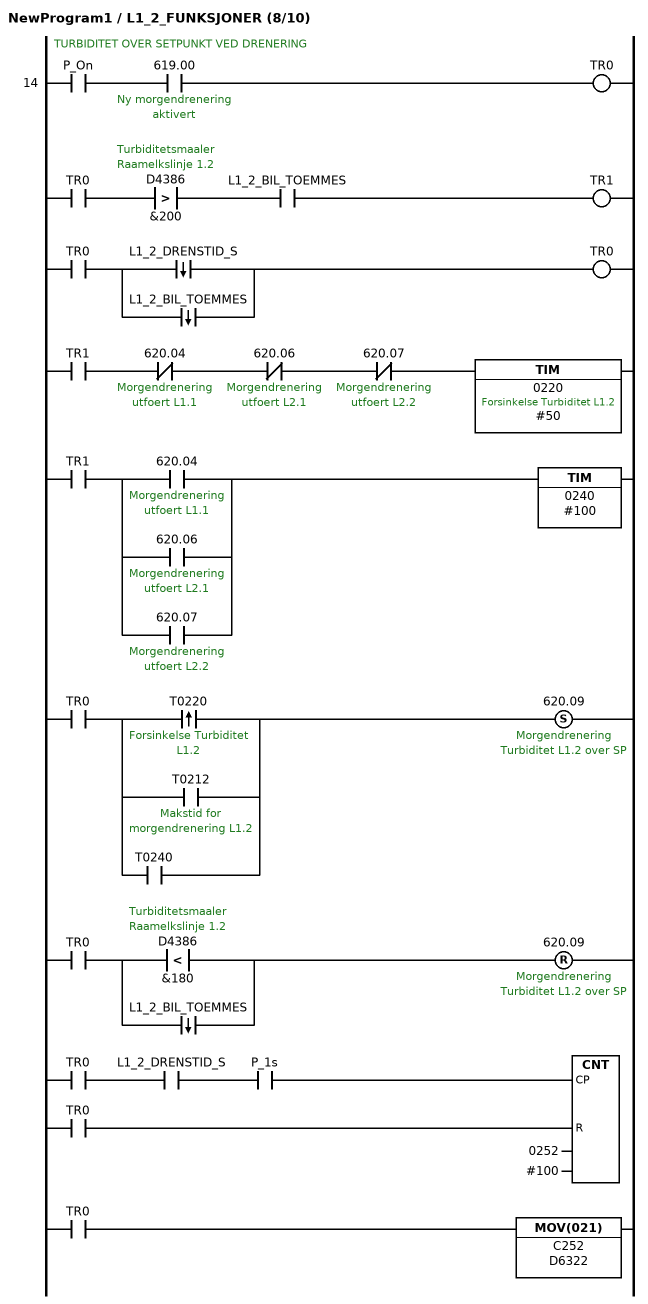
; [picture p792: NewProgram1 / L1_2_FUNKSJONER, rungs 14-14]
; rung 14: TURBIDITET OVER SETPUNKT VED DRENERING
LD P_On
AND 619.00  ; Ny morgendrenering aktivert
OUT TR0
AND>(320) D4386 &200  ; Turbiditetsmaaler Raamelkslinje 1.2
AND L1_2_BIL_TOEMMES
OUT TR1
ANDNOT 620.04  ; Morgendrenering utfoert L1.1
ANDNOT 620.06  ; Morgendrenering utfoert L2.1
ANDNOT 620.07  ; Morgendrenering utfoert L2.2
TIM 0220 #50  ; Forsinkelse Turbiditet L1.2
LD TR1
LD 620.04  ; Morgendrenering utfoert L1.1
OR 620.06  ; Morgendrenering utfoert L2.1
OR 620.07  ; Morgendrenering utfoert L2.2
ANDLD
TIM 0240 #100
LD TR0
@LD T0220  ; Forsinkelse Turbiditet L1.2
OR T0212  ; Makstid for morgendrenering L1.2
OR T0240
ANDLD
SET 620.09  ; Morgendrenering Turbiditet L1.2 over SP
LD TR0
LD<(310) D4386 &180  ; Turbiditetsmaaler Raamelkslinje 1.2
%OR L1_2_BIL_TOEMMES
ANDLD
RSET 620.09  ; Morgendrenering Turbiditet L1.2 over SP
LD TR0
AND L1_2_DRENSTID_S
AND P_1s
LD TR0
%LD L1_2_DRENSTID_S
%OR L1_2_BIL_TOEMMES
ANDLD
OUT TR0
CNT 0252 #100
LD TR0
MOV(021) C252 D6322

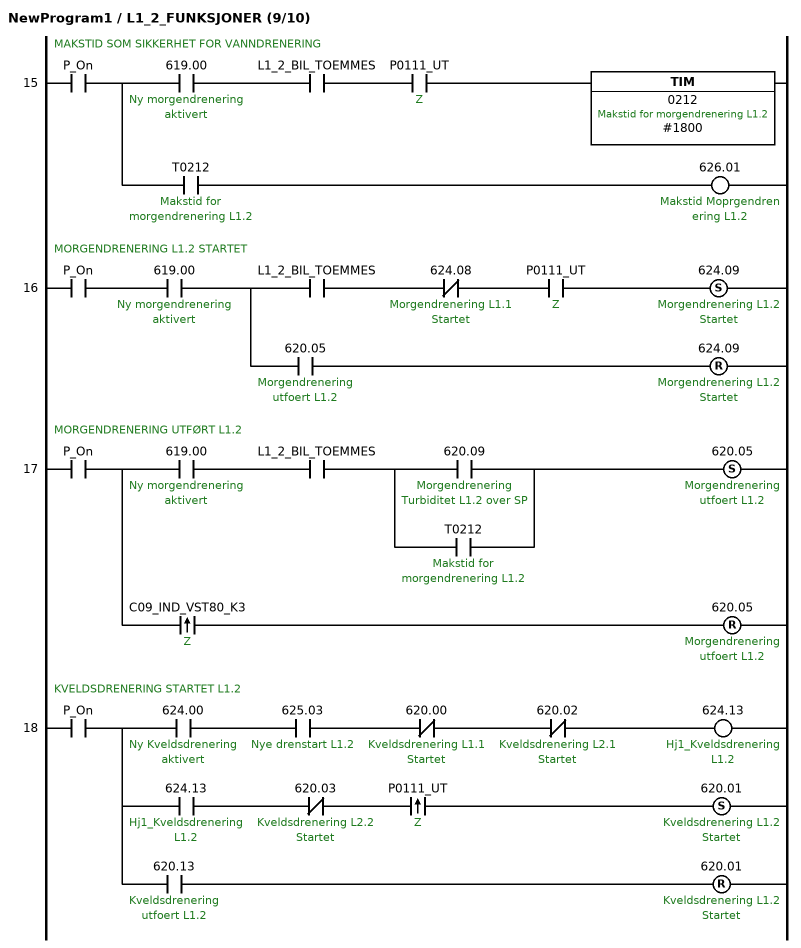
; rung 15: MAKSTID SOM SIKKERHET FOR VANNDRENERING
LD P_On
OUT TR0
AND 619.00  ; Ny morgendrenering aktivert
AND L1_2_BIL_TOEMMES
AND P0111_UT  ; Z
TIM 0212 #1800  ; Makstid for morgendrenering L1.2
LD TR0
AND T0212  ; Makstid for morgendrenering L1.2
OUT 626.01  ; Makstid Moprgendrenering L1.2
; rung 16: MORGENDRENERING L1.2 STARTET
LD P_On
AND 619.00  ; Ny morgendrenering aktivert
OUT TR0
AND L1_2_BIL_TOEMMES
ANDNOT 624.08  ; Morgendrenering L1.1 Startet
AND P0111_UT  ; Z
SET 624.09  ; Morgendrenering L1.2 Startet
LD TR0
AND 620.05  ; Morgendrenering utfoert L1.2
RSET 624.09  ; Morgendrenering L1.2 Startet
; rung 17: MORGENDRENERING UTFØRT L1.2
LD P_On
OUT TR0
AND 619.00  ; Ny morgendrenering aktivert
AND L1_2_BIL_TOEMMES
LD 620.09  ; Morgendrenering Turbiditet L1.2 over SP
OR T0212  ; Makstid for morgendrenering L1.2
ANDLD
SET 620.05  ; Morgendrenering utfoert L1.2
LD TR0
@AND C09_IND_VST80_K3  ; Z
RSET 620.05  ; Morgendrenering utfoert L1.2
; rung 18: KVELDSDRENERING STARTET L1.2
LD P_On
OUT TR0
AND 624.00  ; Ny Kveldsdrenering aktivert
AND 625.03  ; Nye drenstart L1.2
ANDNOT 620.00  ; Kveldsdrenering L1.1 Startet
ANDNOT 620.02  ; Kveldsdrenering L2.1 Startet
OUT 624.13  ; Hj1_Kveldsdrenering L1.2
LD TR0
AND 624.13  ; Hj1_Kveldsdrenering L1.2
ANDNOT 620.03  ; Kveldsdrenering L2.2 Startet
@AND P0111_UT  ; Z
SET 620.01  ; Kveldsdrenering L1.2 Startet
LD TR0
AND 620.13  ; Kveldsdrenering utfoert L1.2
RSET 620.01  ; Kveldsdrenering L1.2 Startet

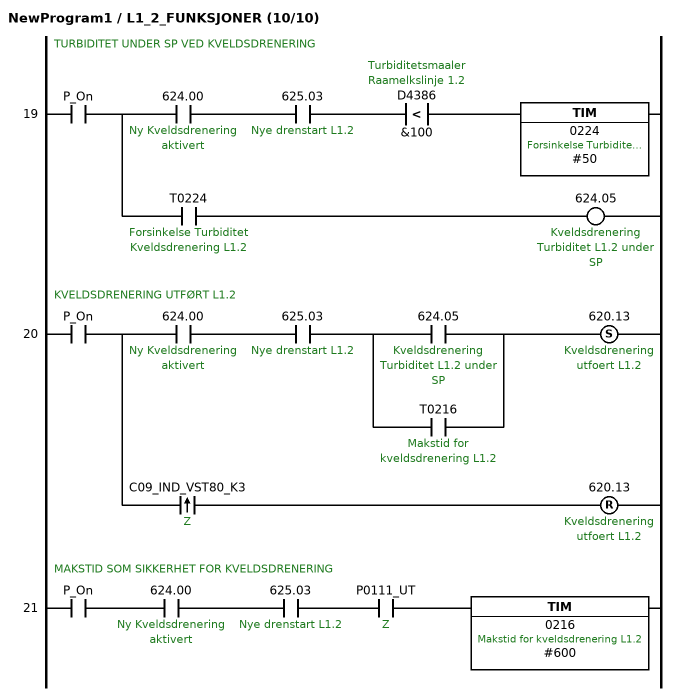
; rung 19: TURBIDITET UNDER SP VED KVELDSDRENERING
LD P_On
OUT TR0
AND 624.00  ; Ny Kveldsdrenering aktivert
AND 625.03  ; Nye drenstart L1.2
AND<(310) D4386 &100  ; Turbiditetsmaaler Raamelkslinje 1.2
TIM 0224 #50  ; Forsinkelse Turbiditet Kveldsdrenering L1.2
LD TR0
AND T0224  ; Forsinkelse Turbiditet Kveldsdrenering L1.2
OUT 624.05  ; Kveldsdrenering Turbiditet L1.2 under SP
; rung 20: KVELDSDRENERING UTFØRT L1.2
LD P_On
OUT TR0
AND 624.00  ; Ny Kveldsdrenering aktivert
AND 625.03  ; Nye drenstart L1.2
LD 624.05  ; Kveldsdrenering Turbiditet L1.2 under SP
OR T0216  ; Makstid for kveldsdrenering L1.2
ANDLD
SET 620.13  ; Kveldsdrenering utfoert L1.2
LD TR0
@AND C09_IND_VST80_K3  ; Z
RSET 620.13  ; Kveldsdrenering utfoert L1.2
; rung 21: MAKSTID SOM SIKKERHET FOR KVELDSDRENERING
LD P_On
AND 624.00  ; Ny Kveldsdrenering aktivert
AND 625.03  ; Nye drenstart L1.2
AND P0111_UT  ; Z
TIM 0216 #600  ; Makstid for kveldsdrenering L1.2
; rung 22: Ingen_kommentar_funnet

### Section L2_1_STATUS

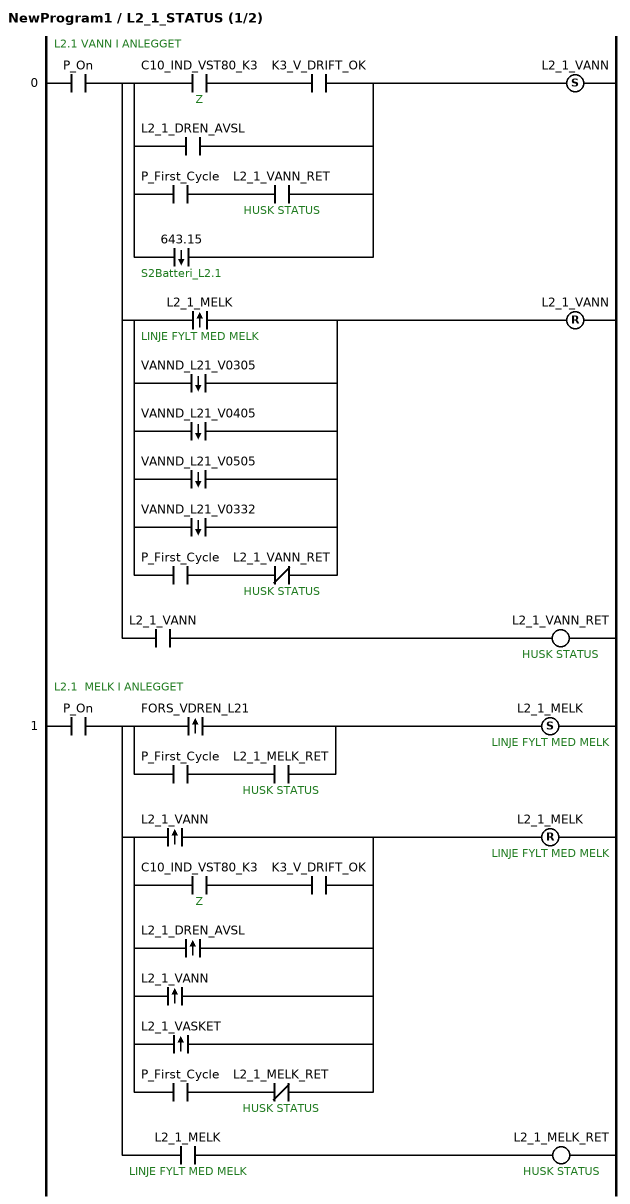
; rung 0: L2.1 VANN I ANLEGGET
LD P_On
OUT TR0
LD C10_IND_VST80_K3  ; Z
AND K3_V_DRIFT_OK
OR L2_1_DREN_AVSL
LD P_First_Cycle
AND L2_1_VANN_RET  ; HUSK STATUS
ORLD
%OR 643.15  ; S2Batteri_L2.1
ANDLD
SET L2_1_VANN
LD TR0
@LD L2_1_MELK  ; LINJE FYLT MED MELK
%OR VANND_L21_V0305
%OR VANND_L21_V0405
%OR VANND_L21_V0505
%OR VANND_L21_V0332
LD P_First_Cycle
ANDNOT L2_1_VANN_RET  ; HUSK STATUS
ORLD
ANDLD
RSET L2_1_VANN
LD TR0
AND L2_1_VANN
OUT L2_1_VANN_RET  ; HUSK STATUS
; rung 1: L2.1  MELK I ANLEGGET
LD P_On
OUT TR0
@LD FORS_VDREN_L21
LD P_First_Cycle
AND L2_1_MELK_RET  ; HUSK STATUS
ORLD
ANDLD
SET L2_1_MELK  ; LINJE FYLT MED MELK
LD TR0
@LD L2_1_VANN
LD C10_IND_VST80_K3  ; Z
AND K3_V_DRIFT_OK
ORLD
@OR L2_1_DREN_AVSL
@OR L2_1_VANN
@OR L2_1_VASKET
LD P_First_Cycle
ANDNOT L2_1_MELK_RET  ; HUSK STATUS
ORLD
ANDLD
RSET L2_1_MELK  ; LINJE FYLT MED MELK
LD TR0
AND L2_1_MELK  ; LINJE FYLT MED MELK
OUT L2_1_MELK_RET  ; HUSK STATUS

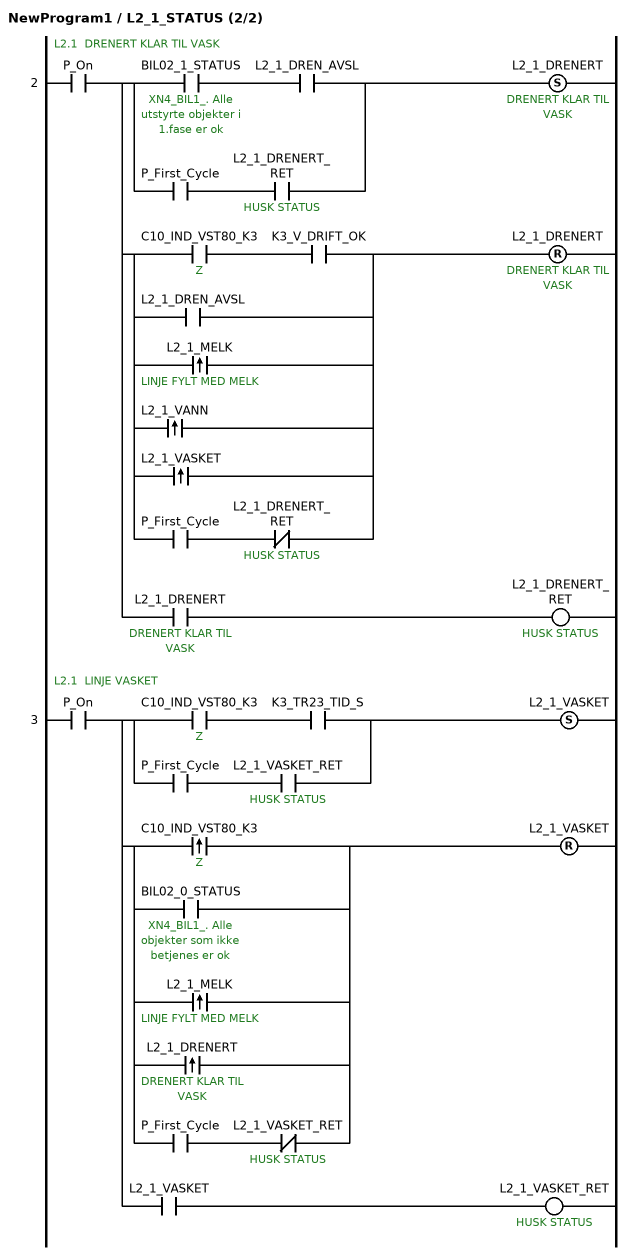
; rung 2: L2.1  DRENERT KLAR TIL VASK
LD P_On
OUT TR0
LD BIL02_1_STATUS  ; XN4_BIL1_. Alle utstyrte objekter i 1.fase er ok
AND L2_1_DREN_AVSL
LD P_First_Cycle
AND L2_1_DRENERT_RET  ; HUSK STATUS
ORLD
ANDLD
SET L2_1_DRENERT  ; DRENERT KLAR TIL VASK
LD TR0
LD C10_IND_VST80_K3  ; Z
AND K3_V_DRIFT_OK
OR L2_1_DREN_AVSL
@OR L2_1_MELK  ; LINJE FYLT MED MELK
@OR L2_1_VANN
@OR L2_1_VASKET
LD P_First_Cycle
ANDNOT L2_1_DRENERT_RET  ; HUSK STATUS
ORLD
ANDLD
RSET L2_1_DRENERT  ; DRENERT KLAR TIL VASK
LD TR0
AND L2_1_DRENERT  ; DRENERT KLAR TIL VASK
OUT L2_1_DRENERT_RET  ; HUSK STATUS
; rung 3: L2.1  LINJE VASKET
LD P_On
OUT TR0
LD C10_IND_VST80_K3  ; Z
AND K3_TR23_TID_S
LD P_First_Cycle
AND L2_1_VASKET_RET  ; HUSK STATUS
ORLD
ANDLD
SET L2_1_VASKET
LD TR0
@LD C10_IND_VST80_K3  ; Z
OR BIL02_0_STATUS  ; XN4_BIL1_. Alle objekter som ikke betjenes er ok
@OR L2_1_MELK  ; LINJE FYLT MED MELK
@OR L2_1_DRENERT  ; DRENERT KLAR TIL VASK
LD P_First_Cycle
ANDNOT L2_1_VASKET_RET  ; HUSK STATUS
ORLD
ANDLD
RSET L2_1_VASKET
LD TR0
AND L2_1_VASKET
OUT L2_1_VASKET_RET  ; HUSK STATUS
; rung 4: Ingen_kommentar_funnet

### Section L1_1_L1_2_FELLESFUNKSJONER

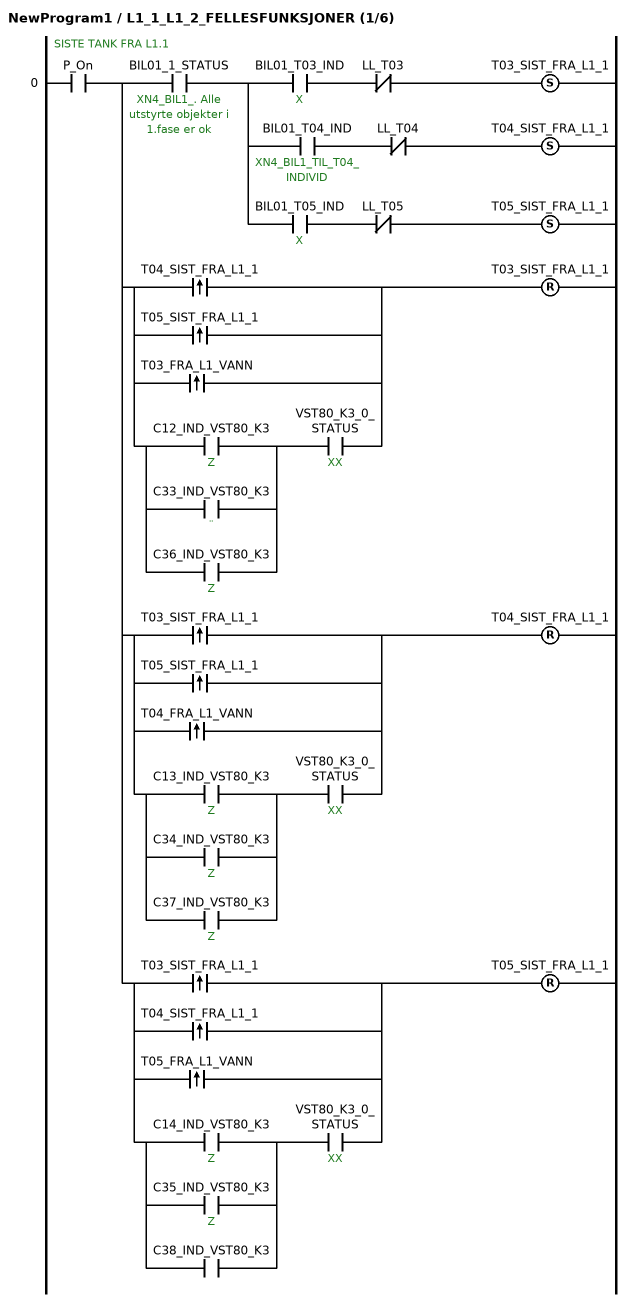
; rung 0: SISTE TANK FRA L1.1
LD P_On
OUT TR0
AND BIL01_1_STATUS  ; XN4_BIL1_. Alle utstyrte objekter i 1.fase er ok
OUT TR1
AND BIL01_T03_IND  ; X
ANDNOT LL_T03
SET T03_SIST_FRA_L1_1
LD TR1
AND BIL01_T04_IND  ; XN4_BIL1_TIL_T04_INDIVID
ANDNOT LL_T04
SET T04_SIST_FRA_L1_1
LD TR1
AND BIL01_T05_IND  ; X
ANDNOT LL_T05
SET T05_SIST_FRA_L1_1
LD TR0
@LD T04_SIST_FRA_L1_1
@OR T05_SIST_FRA_L1_1
@OR T03_FRA_L1_VANN
LD C12_IND_VST80_K3  ; Z
OR C33_IND_VST80_K3  ; ¨
OR C36_IND_VST80_K3  ; Z
AND VST80_K3_0_STATUS  ; XX
ORLD
ANDLD
RSET T03_SIST_FRA_L1_1
LD TR0
@LD T03_SIST_FRA_L1_1
@OR T05_SIST_FRA_L1_1
@OR T04_FRA_L1_VANN
LD C13_IND_VST80_K3  ; Z
OR C34_IND_VST80_K3  ; Z
OR C37_IND_VST80_K3  ; Z
AND VST80_K3_0_STATUS  ; XX
ORLD
ANDLD
RSET T04_SIST_FRA_L1_1
LD TR0
@LD T03_SIST_FRA_L1_1
@OR T04_SIST_FRA_L1_1
@OR T05_FRA_L1_VANN
LD C14_IND_VST80_K3  ; Z
OR C35_IND_VST80_K3  ; Z
OR C38_IND_VST80_K3
AND VST80_K3_0_STATUS  ; XX
ORLD
ANDLD
RSET T05_SIST_FRA_L1_1

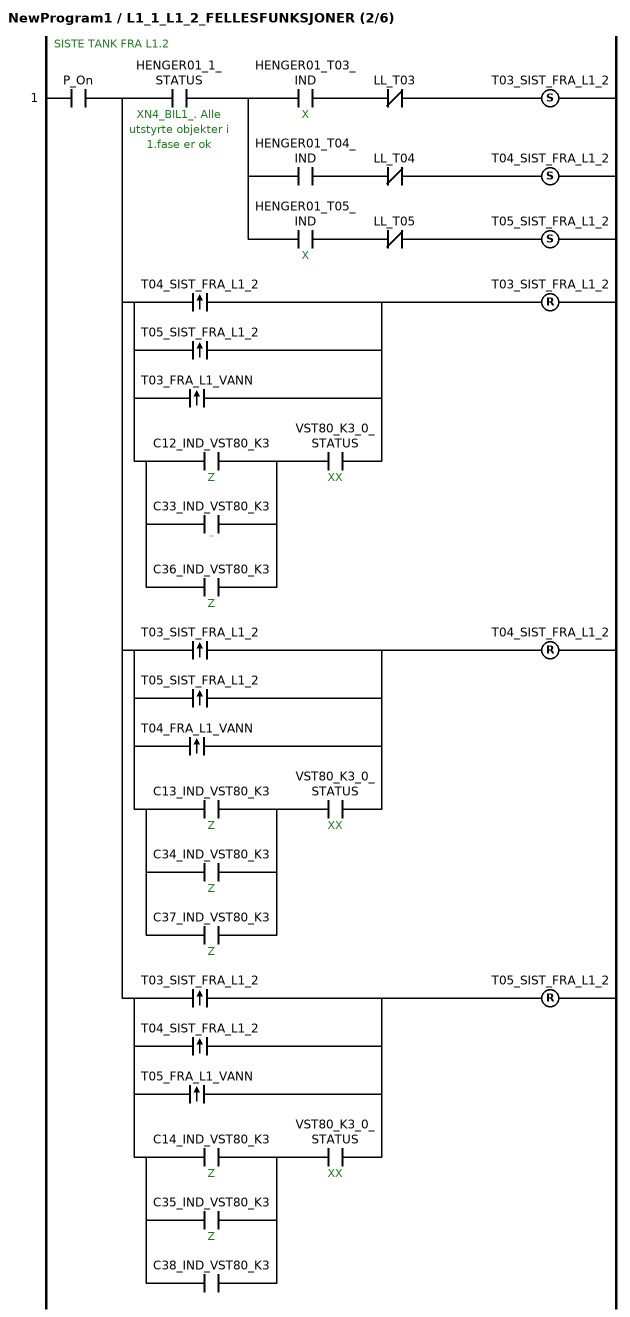
; rung 1: SISTE TANK FRA L1.2
LD P_On
OUT TR0
AND HENGER01_1_STATUS  ; XN4_BIL1_. Alle utstyrte objekter i 1.fase er ok
OUT TR1
AND HENGER01_T03_IND  ; X
ANDNOT LL_T03
SET T03_SIST_FRA_L1_2
LD TR1
AND HENGER01_T04_IND
ANDNOT LL_T04
SET T04_SIST_FRA_L1_2
LD TR1
AND HENGER01_T05_IND  ; X
ANDNOT LL_T05
SET T05_SIST_FRA_L1_2
LD TR0
@LD T04_SIST_FRA_L1_2
@OR T05_SIST_FRA_L1_2
@OR T03_FRA_L1_VANN
LD C12_IND_VST80_K3  ; Z
OR C33_IND_VST80_K3  ; ¨
OR C36_IND_VST80_K3  ; Z
AND VST80_K3_0_STATUS  ; XX
ORLD
ANDLD
RSET T03_SIST_FRA_L1_2
LD TR0
@LD T03_SIST_FRA_L1_2
@OR T05_SIST_FRA_L1_2
@OR T04_FRA_L1_VANN
LD C13_IND_VST80_K3  ; Z
OR C34_IND_VST80_K3  ; Z
OR C37_IND_VST80_K3  ; Z
AND VST80_K3_0_STATUS  ; XX
ORLD
ANDLD
RSET T04_SIST_FRA_L1_2
LD TR0
@LD T03_SIST_FRA_L1_2
@OR T04_SIST_FRA_L1_2
@OR T05_FRA_L1_VANN
LD C14_IND_VST80_K3  ; Z
OR C35_IND_VST80_K3  ; Z
OR C38_IND_VST80_K3
AND VST80_K3_0_STATUS  ; XX
ORLD
ANDLD
RSET T05_SIST_FRA_L1_2

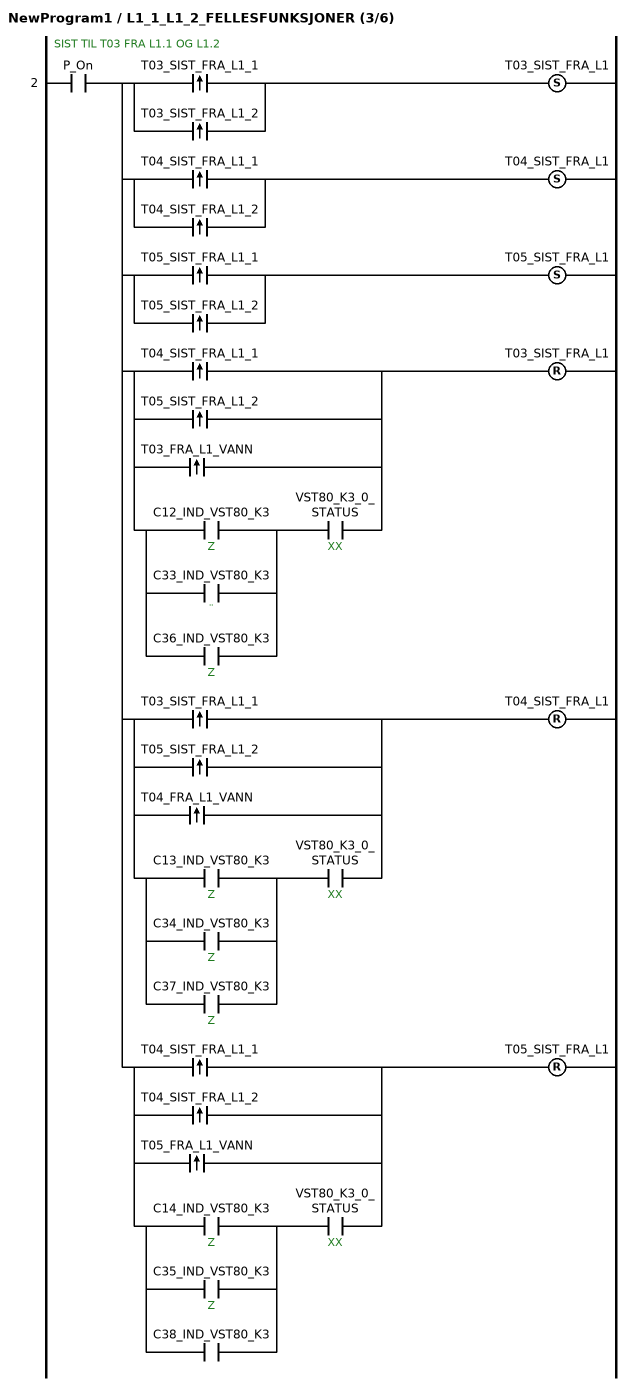
; rung 2: SIST TIL T03 FRA L1.1 OG L1.2
LD P_On
OUT TR0
@LD T03_SIST_FRA_L1_1
@OR T03_SIST_FRA_L1_2
ANDLD
SET T03_SIST_FRA_L1
LD TR0
@LD T04_SIST_FRA_L1_1
@OR T04_SIST_FRA_L1_2
ANDLD
SET T04_SIST_FRA_L1
LD TR0
@LD T05_SIST_FRA_L1_1
@OR T05_SIST_FRA_L1_2
ANDLD
SET T05_SIST_FRA_L1
LD TR0
@LD T04_SIST_FRA_L1_1
@OR T05_SIST_FRA_L1_2
@OR T03_FRA_L1_VANN
LD C12_IND_VST80_K3  ; Z
OR C33_IND_VST80_K3  ; ¨
OR C36_IND_VST80_K3  ; Z
AND VST80_K3_0_STATUS  ; XX
ORLD
ANDLD
RSET T03_SIST_FRA_L1
LD TR0
@LD T03_SIST_FRA_L1_1
@OR T05_SIST_FRA_L1_2
@OR T04_FRA_L1_VANN
LD C13_IND_VST80_K3  ; Z
OR C34_IND_VST80_K3  ; Z
OR C37_IND_VST80_K3  ; Z
AND VST80_K3_0_STATUS  ; XX
ORLD
ANDLD
RSET T04_SIST_FRA_L1
LD TR0
@LD T04_SIST_FRA_L1_1
@OR T04_SIST_FRA_L1_2
@OR T05_FRA_L1_VANN
LD C14_IND_VST80_K3  ; Z
OR C35_IND_VST80_K3  ; Z
OR C38_IND_VST80_K3
AND VST80_K3_0_STATUS  ; XX
ORLD
ANDLD
RSET T05_SIST_FRA_L1

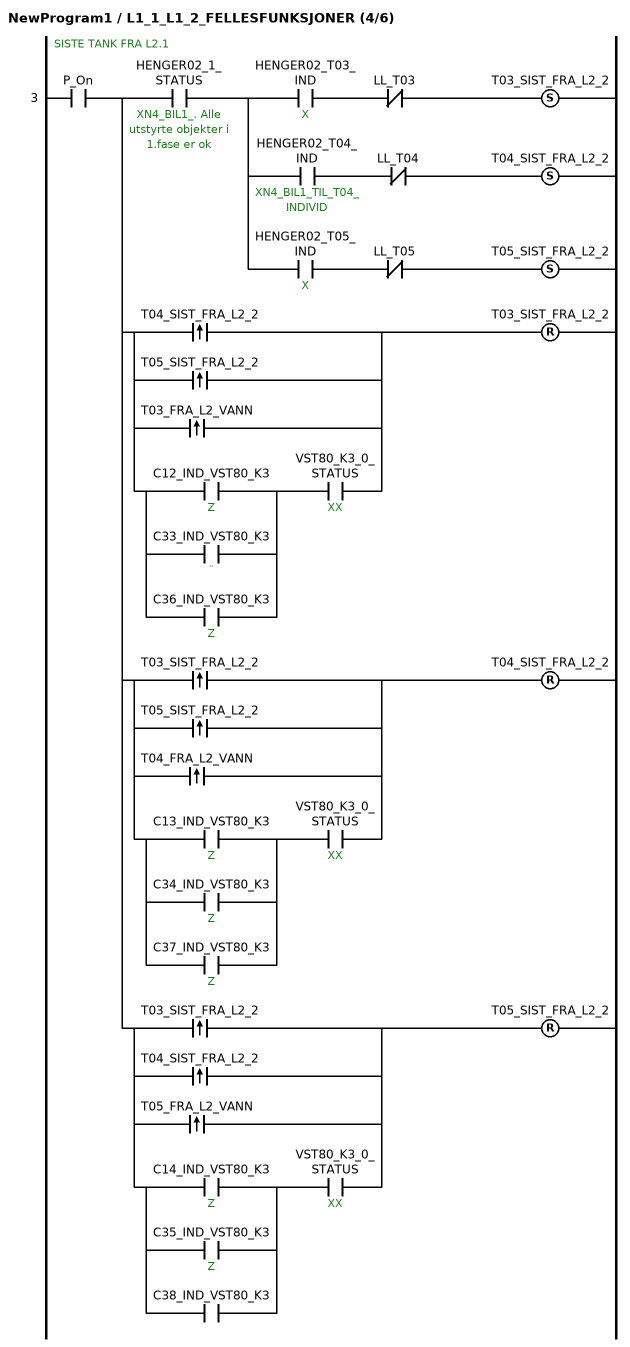
; rung 3: SISTE TANK FRA L2.1
LD P_On
OUT TR0
AND HENGER02_1_STATUS  ; XN4_BIL1_. Alle utstyrte objekter i 1.fase er ok
OUT TR1
AND HENGER02_T03_IND  ; X
ANDNOT LL_T03
SET T03_SIST_FRA_L2_2
LD TR1
AND HENGER02_T04_IND  ; XN4_BIL1_TIL_T04_INDIVID
ANDNOT LL_T04
SET T04_SIST_FRA_L2_2
LD TR1
AND HENGER02_T05_IND  ; X
ANDNOT LL_T05
SET T05_SIST_FRA_L2_2
LD TR0
@LD T04_SIST_FRA_L2_2
@OR T05_SIST_FRA_L2_2
@OR T03_FRA_L2_VANN
LD C12_IND_VST80_K3  ; Z
OR C33_IND_VST80_K3  ; ¨
OR C36_IND_VST80_K3  ; Z
AND VST80_K3_0_STATUS  ; XX
ORLD
ANDLD
RSET T03_SIST_FRA_L2_2
LD TR0
@LD T03_SIST_FRA_L2_2
@OR T05_SIST_FRA_L2_2
@OR T04_FRA_L2_VANN
LD C13_IND_VST80_K3  ; Z
OR C34_IND_VST80_K3  ; Z
OR C37_IND_VST80_K3  ; Z
AND VST80_K3_0_STATUS  ; XX
ORLD
ANDLD
RSET T04_SIST_FRA_L2_2
LD TR0
@LD T03_SIST_FRA_L2_2
@OR T04_SIST_FRA_L2_2
@OR T05_FRA_L2_VANN
LD C14_IND_VST80_K3  ; Z
OR C35_IND_VST80_K3  ; Z
OR C38_IND_VST80_K3
AND VST80_K3_0_STATUS  ; XX
ORLD
ANDLD
RSET T05_SIST_FRA_L2_2

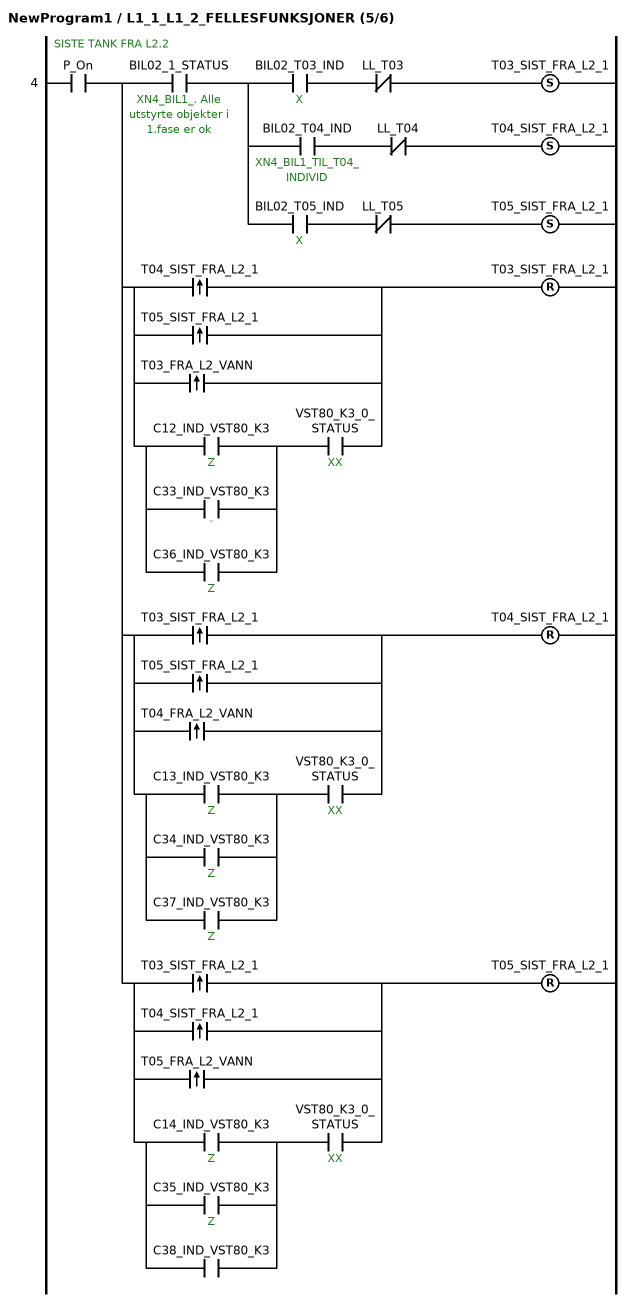
; rung 4: SISTE TANK FRA L2.2
LD P_On
OUT TR0
AND BIL02_1_STATUS  ; XN4_BIL1_. Alle utstyrte objekter i 1.fase er ok
OUT TR1
AND BIL02_T03_IND  ; X
ANDNOT LL_T03
SET T03_SIST_FRA_L2_1
LD TR1
AND BIL02_T04_IND  ; XN4_BIL1_TIL_T04_INDIVID
ANDNOT LL_T04
SET T04_SIST_FRA_L2_1
LD TR1
AND BIL02_T05_IND  ; X
ANDNOT LL_T05
SET T05_SIST_FRA_L2_1
LD TR0
@LD T04_SIST_FRA_L2_1
@OR T05_SIST_FRA_L2_1
@OR T03_FRA_L2_VANN
LD C12_IND_VST80_K3  ; Z
OR C33_IND_VST80_K3  ; ¨
OR C36_IND_VST80_K3  ; Z
AND VST80_K3_0_STATUS  ; XX
ORLD
ANDLD
RSET T03_SIST_FRA_L2_1
LD TR0
@LD T03_SIST_FRA_L2_1
@OR T05_SIST_FRA_L2_1
@OR T04_FRA_L2_VANN
LD C13_IND_VST80_K3  ; Z
OR C34_IND_VST80_K3  ; Z
OR C37_IND_VST80_K3  ; Z
AND VST80_K3_0_STATUS  ; XX
ORLD
ANDLD
RSET T04_SIST_FRA_L2_1
LD TR0
@LD T03_SIST_FRA_L2_1
@OR T04_SIST_FRA_L2_1
@OR T05_FRA_L2_VANN
LD C14_IND_VST80_K3  ; Z
OR C35_IND_VST80_K3  ; Z
OR C38_IND_VST80_K3
AND VST80_K3_0_STATUS  ; XX
ORLD
ANDLD
RSET T05_SIST_FRA_L2_1

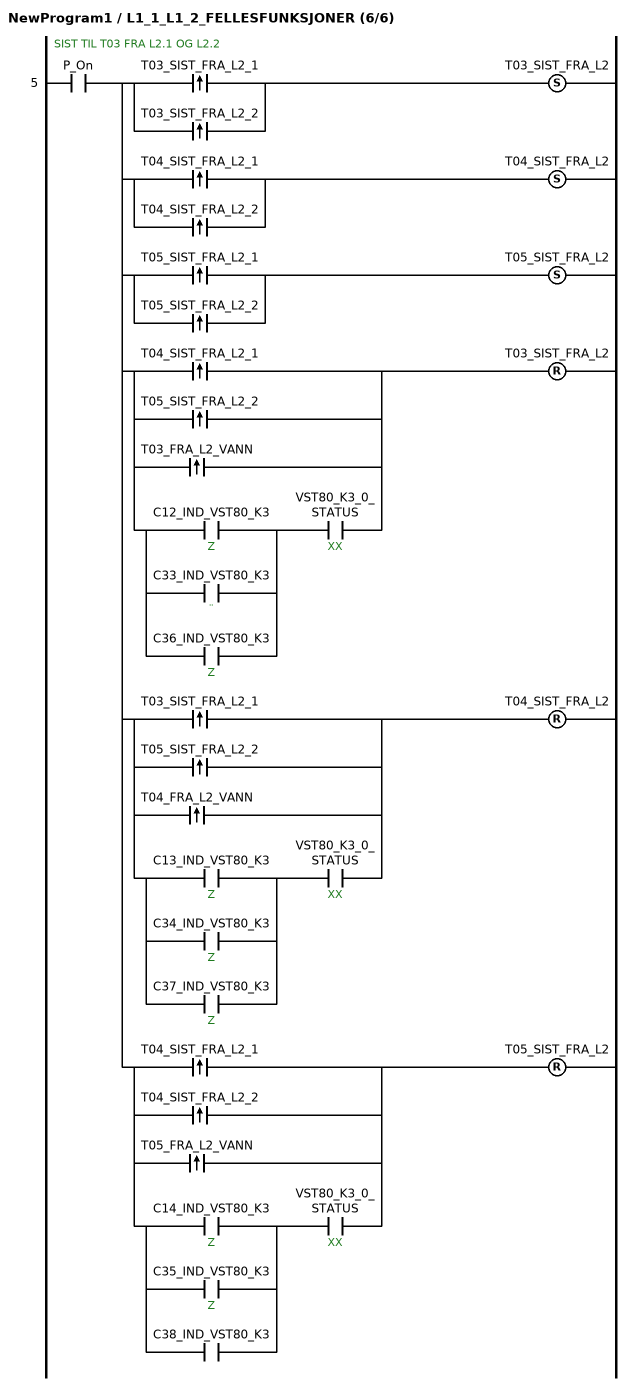
; rung 5: SIST TIL T03 FRA L2.1 OG L2.2
LD P_On
OUT TR0
@LD T03_SIST_FRA_L2_1
@OR T03_SIST_FRA_L2_2
ANDLD
SET T03_SIST_FRA_L2
LD TR0
@LD T04_SIST_FRA_L2_1
@OR T04_SIST_FRA_L2_2
ANDLD
SET T04_SIST_FRA_L2
LD TR0
@LD T05_SIST_FRA_L2_1
@OR T05_SIST_FRA_L2_2
ANDLD
SET T05_SIST_FRA_L2
LD TR0
@LD T04_SIST_FRA_L2_1
@OR T05_SIST_FRA_L2_2
@OR T03_FRA_L2_VANN
LD C12_IND_VST80_K3  ; Z
OR C33_IND_VST80_K3  ; ¨
OR C36_IND_VST80_K3  ; Z
AND VST80_K3_0_STATUS  ; XX
ORLD
ANDLD
RSET T03_SIST_FRA_L2
LD TR0
@LD T03_SIST_FRA_L2_1
@OR T05_SIST_FRA_L2_2
@OR T04_FRA_L2_VANN
LD C13_IND_VST80_K3  ; Z
OR C34_IND_VST80_K3  ; Z
OR C37_IND_VST80_K3  ; Z
AND VST80_K3_0_STATUS  ; XX
ORLD
ANDLD
RSET T04_SIST_FRA_L2
LD TR0
@LD T04_SIST_FRA_L2_1
@OR T04_SIST_FRA_L2_2
@OR T05_FRA_L2_VANN
LD C14_IND_VST80_K3  ; Z
OR C35_IND_VST80_K3  ; Z
OR C38_IND_VST80_K3
AND VST80_K3_0_STATUS  ; XX
ORLD
ANDLD
RSET T05_SIST_FRA_L2
; rung 6: Ingen_kommentar_funnet

### Section L2_1_FUNKSJONER

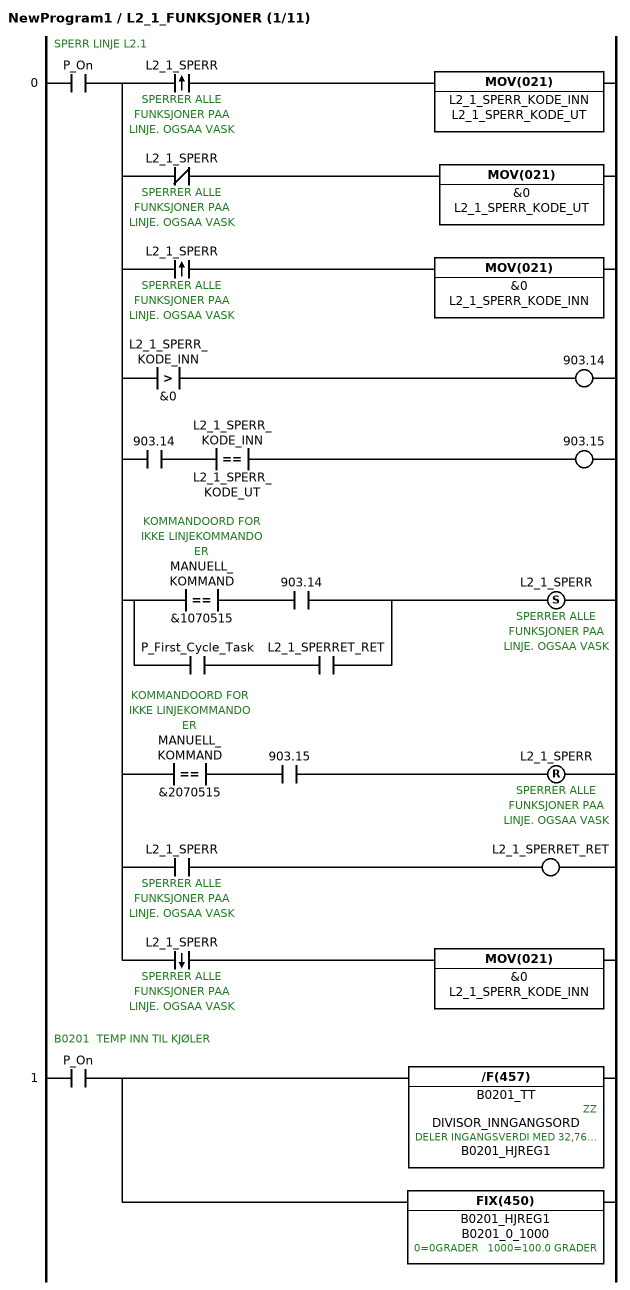
; rung 0: SPERR LINJE L2.1
LD P_On
OUT TR0
@AND L2_1_SPERR  ; SPERRER ALLE FUNKSJONER PAA LINJE. OGSAA VASK
MOV(021) L2_1_SPERR_KODE_INN L2_1_SPERR_KODE_UT
LD TR0
ANDNOT L2_1_SPERR  ; SPERRER ALLE FUNKSJONER PAA LINJE. OGSAA VASK
MOV(021) &0 L2_1_SPERR_KODE_UT
LD TR0
@AND L2_1_SPERR  ; SPERRER ALLE FUNKSJONER PAA LINJE. OGSAA VASK
MOV(021) &0 L2_1_SPERR_KODE_INN
LD TR0
AND>(320) L2_1_SPERR_KODE_INN &0
OUT 903.14
LD TR0
AND 903.14
AND=(300) L2_1_SPERR_KODE_INN L2_1_SPERR_KODE_UT
OUT 903.15
LD TR0
LD=L(301) MANUELL_KOMMAND &1070515  ; KOMMANDOORD FOR IKKE LINJEKOMMANDOER
AND 903.14
LD P_First_Cycle_Task
AND L2_1_SPERRET_RET
ORLD
ANDLD
SET L2_1_SPERR  ; SPERRER ALLE FUNKSJONER PAA LINJE. OGSAA VASK
LD TR0
AND=L(301) MANUELL_KOMMAND &2070515  ; KOMMANDOORD FOR IKKE LINJEKOMMANDOER
AND 903.15
RSET L2_1_SPERR  ; SPERRER ALLE FUNKSJONER PAA LINJE. OGSAA VASK
LD TR0
AND L2_1_SPERR  ; SPERRER ALLE FUNKSJONER PAA LINJE. OGSAA VASK
OUT L2_1_SPERRET_RET
LD TR0
%AND L2_1_SPERR  ; SPERRER ALLE FUNKSJONER PAA LINJE. OGSAA VASK
MOV(021) &0 L2_1_SPERR_KODE_INN
; rung 1: B0201  TEMP INN TIL KJØLER
LD P_On
/F(457) B0201_TT DIVISOR_INNGANGSORD B0201_HJREG1  ; ZZ, DELER INGANGSVERDI MED 32,760 FOR OMREGNING TIL 0-1000
FIX(450) B0201_HJREG1 B0201_0_1000  ; 0=0GRADER   1000=100.0 GRADER

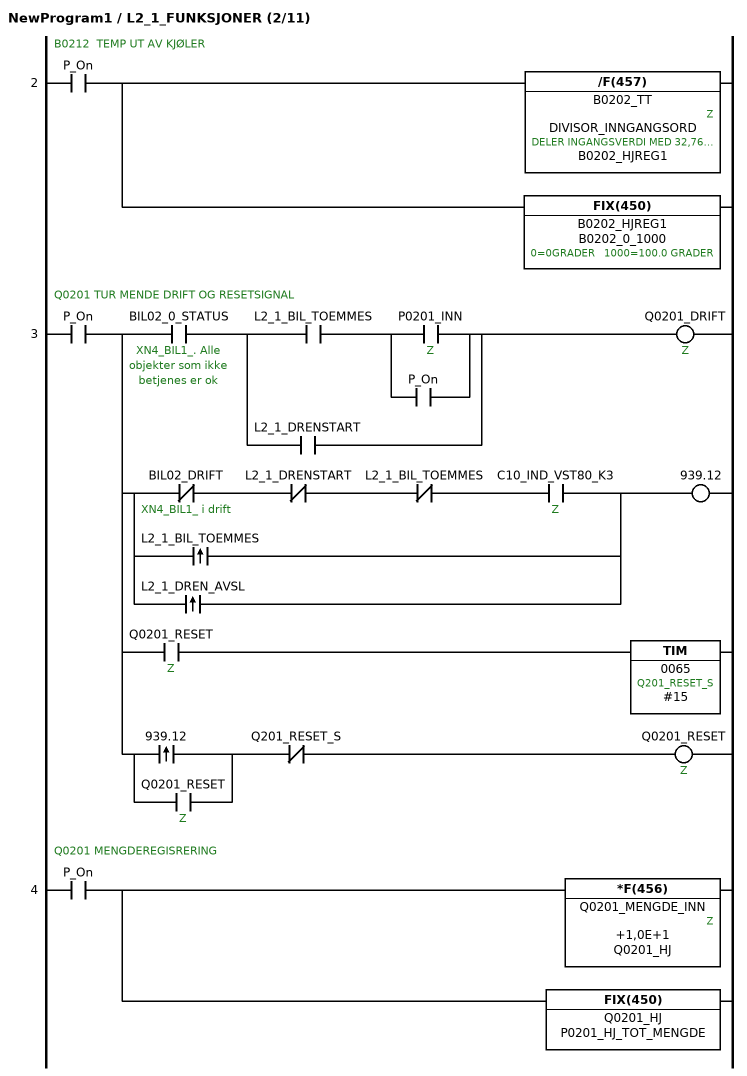
; rung 2: B0212  TEMP UT AV KJØLER
LD P_On
/F(457) B0202_TT DIVISOR_INNGANGSORD B0202_HJREG1  ; Z, DELER INGANGSVERDI MED 32,760 FOR OMREGNING TIL 0-1000
FIX(450) B0202_HJREG1 B0202_0_1000  ; 0=0GRADER   1000=100.0 GRADER
; rung 3: Q0201 TUR MENDE DRIFT OG RESETSIGNAL
LD P_On
OUT TR0
AND BIL02_0_STATUS  ; XN4_BIL1_. Alle objekter som ikke betjenes er ok
LD L2_1_BIL_TOEMMES
LD P0201_INN  ; Z
OR P_On
ANDLD
OR L2_1_DRENSTART
ANDLD
OUT Q0201_DRIFT  ; Z
LD TR0
LDNOT BIL02_DRIFT  ; XN4_BIL1_ i drift
ANDNOT L2_1_DRENSTART
ANDNOT L2_1_BIL_TOEMMES
AND C10_IND_VST80_K3  ; Z
@OR L2_1_BIL_TOEMMES
@OR L2_1_DREN_AVSL
ANDLD
OUT 939.12
LD TR0
AND Q0201_RESET  ; Z
TIM 0065 #15  ; Q201_RESET_S
LD TR0
@LD 939.12
OR Q0201_RESET  ; Z
ANDLD
ANDNOT Q201_RESET_S
OUT Q0201_RESET  ; Z
; rung 4: Q0201 MENGDEREGISRERING
LD P_On
*F(456) Q0201_MENGDE_INN +1,0E+1 Q0201_HJ  ; Z
FIX(450) Q0201_HJ P0201_HJ_TOT_MENGDE

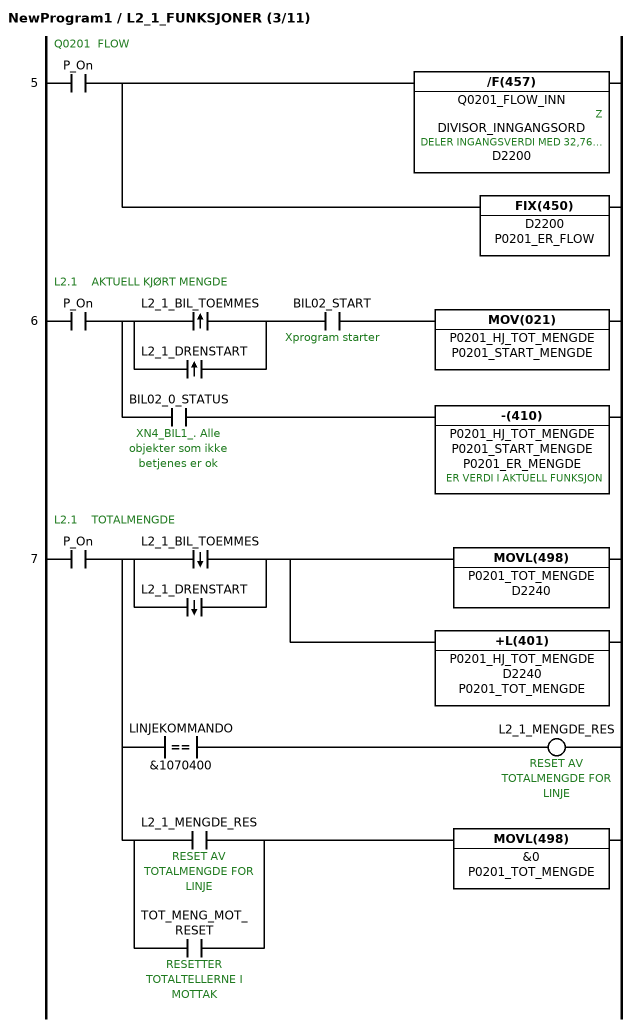
; rung 5: Q0201  FLOW
LD P_On
/F(457) Q0201_FLOW_INN DIVISOR_INNGANGSORD D2200  ; Z, DELER INGANGSVERDI MED 32,760 FOR OMREGNING TIL 0-1000
FIX(450) D2200 P0201_ER_FLOW
; rung 6: L2.1    AKTUELL KJØRT MENGDE
LD P_On
OUT TR0
@LD L2_1_BIL_TOEMMES
@OR L2_1_DRENSTART
ANDLD
AND BIL02_START  ; Xprogram starter
MOV(021) P0201_HJ_TOT_MENGDE P0201_START_MENGDE
LD TR0
AND BIL02_0_STATUS  ; XN4_BIL1_. Alle objekter som ikke betjenes er ok
-(410) P0201_HJ_TOT_MENGDE P0201_START_MENGDE P0201_ER_MENGDE  ; ER VERDI I AKTUELL FUNKSJON
; rung 7: L2.1    TOTALMENGDE
LD P_On
OUT TR0
%LD L2_1_BIL_TOEMMES
%OR L2_1_DRENSTART
ANDLD
MOVL(498) P0201_TOT_MENGDE D2240
+L(401) P0201_HJ_TOT_MENGDE D2240 P0201_TOT_MENGDE
LD TR0
AND=L(301) LINJEKOMMANDO &1070400
OUT L2_1_MENGDE_RES  ; RESET AV  TOTALMENGDE FOR LINJE
LD TR0
LD L2_1_MENGDE_RES  ; RESET AV  TOTALMENGDE FOR LINJE
OR TOT_MENG_MOT_RESET  ; RESETTER TOTALTELLERNE I MOTTAK
ANDLD
MOVL(498) &0 P0201_TOT_MENGDE

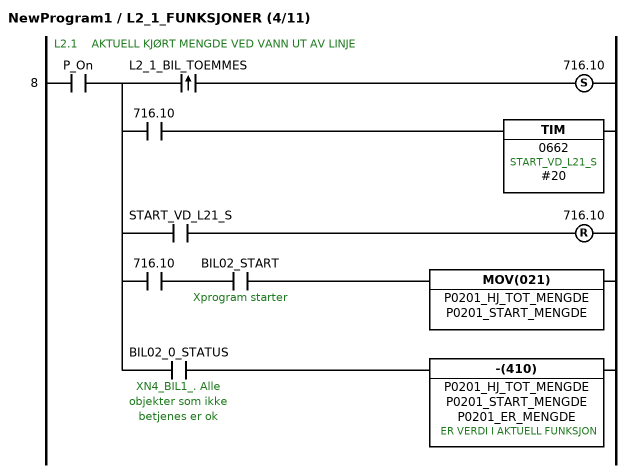
; rung 8: L2.1    AKTUELL KJØRT MENGDE VED VANN UT AV LINJE
LD P_On
OUT TR0
@AND L2_1_BIL_TOEMMES
SET 716.10
LD TR0
AND 716.10
TIM 0662 #20  ; START_VD_L21_S
LD TR0
AND START_VD_L21_S
RSET 716.10
LD TR0
AND 716.10
AND BIL02_START  ; Xprogram starter
MOV(021) P0201_HJ_TOT_MENGDE P0201_START_MENGDE
LD TR0
AND BIL02_0_STATUS  ; XN4_BIL1_. Alle objekter som ikke betjenes er ok
-(410) P0201_HJ_TOT_MENGDE P0201_START_MENGDE P0201_ER_MENGDE  ; ER VERDI I AKTUELL FUNKSJON

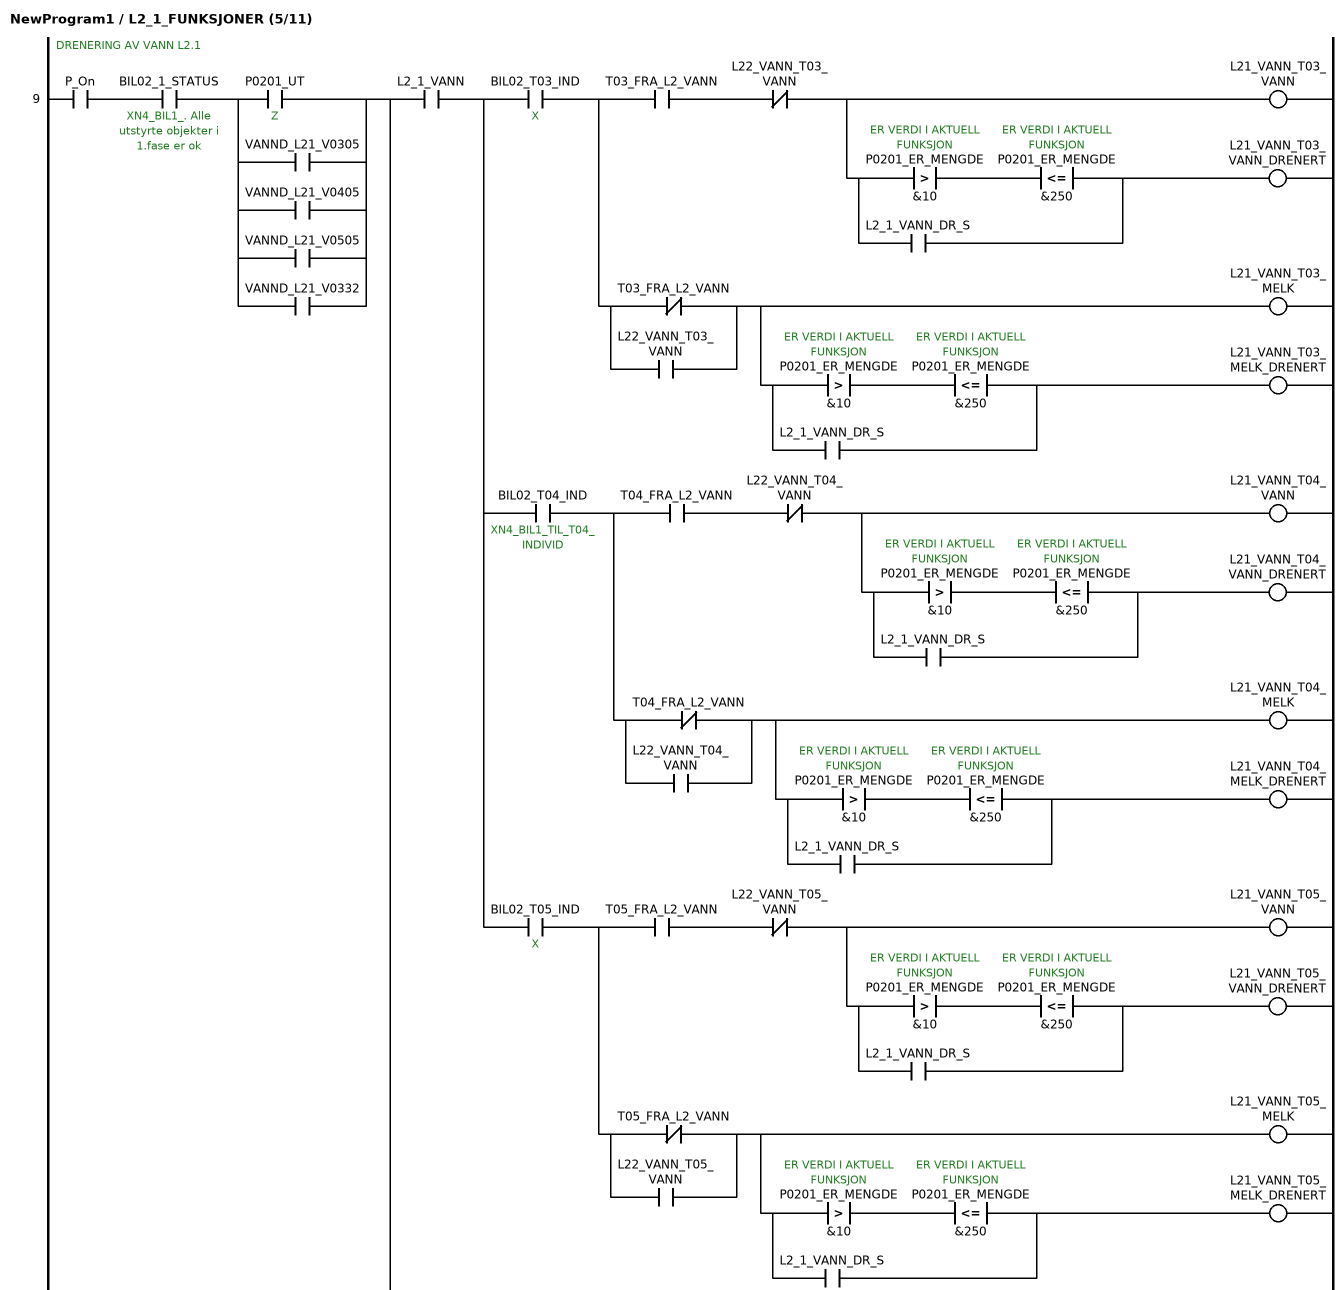

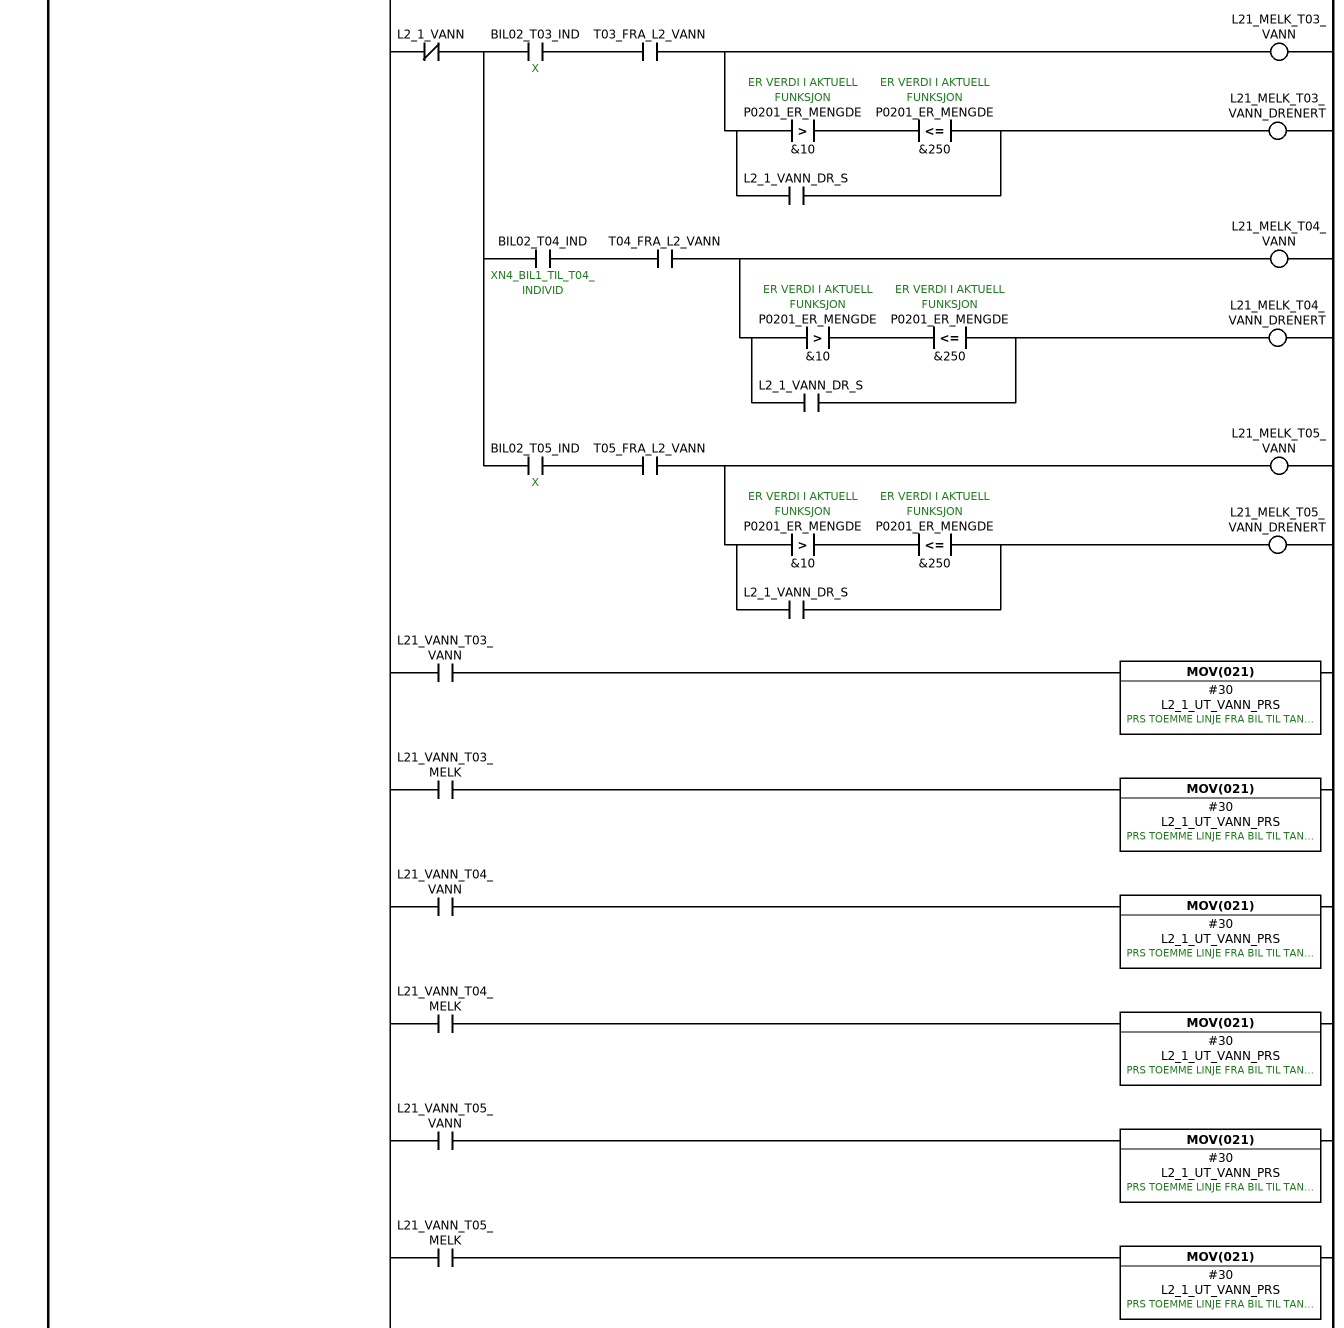

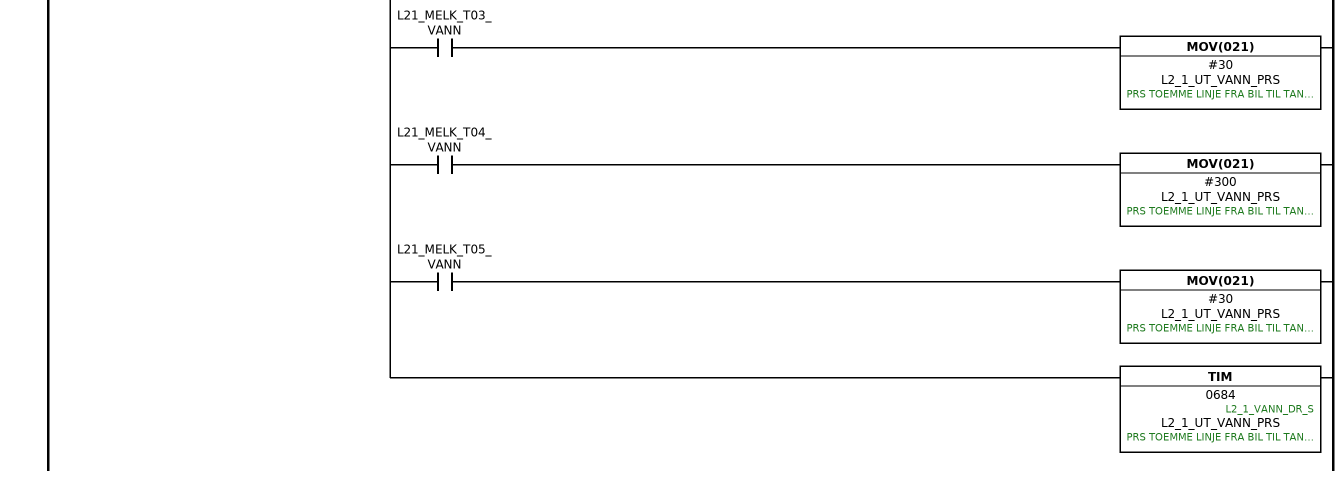
; rung 9: DRENERING AV VANN L2.1
LD P_On
AND BIL02_1_STATUS  ; XN4_BIL1_. Alle utstyrte objekter i 1.fase er ok
LD P0201_UT  ; Z
OR VANND_L21_V0305
OR VANND_L21_V0405
OR VANND_L21_V0505
OR VANND_L21_V0332
ANDLD
OUT TR0
AND L2_1_VANN
OUT TR1
AND BIL02_T03_IND  ; X
OUT TR2
AND T03_FRA_L2_VANN
ANDNOT L22_VANN_T03_VANN
OUT L21_VANN_T03_VANN
LD>(320) P0201_ER_MENGDE &10  ; ER VERDI I AKTUELL FUNKSJON
AND<=(315) P0201_ER_MENGDE &250  ; ER VERDI I AKTUELL FUNKSJON
OR L2_1_VANN_DR_S
ANDLD
OUT L21_VANN_T03_VANN_DRENERT
LD TR2
LDNOT T03_FRA_L2_VANN
OR L22_VANN_T03_VANN
ANDLD
OUT L21_VANN_T03_MELK
LD>(320) P0201_ER_MENGDE &10  ; ER VERDI I AKTUELL FUNKSJON
AND<=(315) P0201_ER_MENGDE &250  ; ER VERDI I AKTUELL FUNKSJON
OR L2_1_VANN_DR_S
ANDLD
OUT L21_VANN_T03_MELK_DRENERT
LD TR1
AND BIL02_T04_IND  ; XN4_BIL1_TIL_T04_INDIVID
OUT TR2
AND T04_FRA_L2_VANN
ANDNOT L22_VANN_T04_VANN
OUT L21_VANN_T04_VANN
LD>(320) P0201_ER_MENGDE &10  ; ER VERDI I AKTUELL FUNKSJON
AND<=(315) P0201_ER_MENGDE &250  ; ER VERDI I AKTUELL FUNKSJON
OR L2_1_VANN_DR_S
ANDLD
OUT L21_VANN_T04_VANN_DRENERT
LD TR2
LDNOT T04_FRA_L2_VANN
OR L22_VANN_T04_VANN
ANDLD
OUT L21_VANN_T04_MELK
LD>(320) P0201_ER_MENGDE &10  ; ER VERDI I AKTUELL FUNKSJON
AND<=(315) P0201_ER_MENGDE &250  ; ER VERDI I AKTUELL FUNKSJON
OR L2_1_VANN_DR_S
ANDLD
OUT L21_VANN_T04_MELK_DRENERT
LD TR1
AND BIL02_T05_IND  ; X
OUT TR1
AND T05_FRA_L2_VANN
ANDNOT L22_VANN_T05_VANN
OUT L21_VANN_T05_VANN
LD>(320) P0201_ER_MENGDE &10  ; ER VERDI I AKTUELL FUNKSJON
AND<=(315) P0201_ER_MENGDE &250  ; ER VERDI I AKTUELL FUNKSJON
OR L2_1_VANN_DR_S
ANDLD
OUT L21_VANN_T05_VANN_DRENERT
LD TR1
LDNOT T05_FRA_L2_VANN
OR L22_VANN_T05_VANN
ANDLD
OUT L21_VANN_T05_MELK
LD>(320) P0201_ER_MENGDE &10  ; ER VERDI I AKTUELL FUNKSJON
AND<=(315) P0201_ER_MENGDE &250  ; ER VERDI I AKTUELL FUNKSJON
OR L2_1_VANN_DR_S
ANDLD
OUT L21_VANN_T05_MELK_DRENERT
LD TR0
ANDNOT L2_1_VANN
OUT TR1
AND BIL02_T03_IND  ; X
AND T03_FRA_L2_VANN
OUT L21_MELK_T03_VANN
LD>(320) P0201_ER_MENGDE &10  ; ER VERDI I AKTUELL FUNKSJON
AND<=(315) P0201_ER_MENGDE &250  ; ER VERDI I AKTUELL FUNKSJON
OR L2_1_VANN_DR_S
ANDLD
OUT L21_MELK_T03_VANN_DRENERT
LD TR1
AND BIL02_T04_IND  ; XN4_BIL1_TIL_T04_INDIVID
AND T04_FRA_L2_VANN
OUT L21_MELK_T04_VANN
LD>(320) P0201_ER_MENGDE &10  ; ER VERDI I AKTUELL FUNKSJON
AND<=(315) P0201_ER_MENGDE &250  ; ER VERDI I AKTUELL FUNKSJON
OR L2_1_VANN_DR_S
ANDLD
OUT L21_MELK_T04_VANN_DRENERT
LD TR1
AND BIL02_T05_IND  ; X
AND T05_FRA_L2_VANN
OUT L21_MELK_T05_VANN
LD>(320) P0201_ER_MENGDE &10  ; ER VERDI I AKTUELL FUNKSJON
AND<=(315) P0201_ER_MENGDE &250  ; ER VERDI I AKTUELL FUNKSJON
OR L2_1_VANN_DR_S
ANDLD
OUT L21_MELK_T05_VANN_DRENERT
LD TR0
AND L21_VANN_T03_VANN
MOV(021) #30 L2_1_UT_VANN_PRS  ; PRS TOEMME LINJE FRA BIL TIL TANK FOR VANN
LD TR0
AND L21_VANN_T03_MELK
MOV(021) #30 L2_1_UT_VANN_PRS  ; PRS TOEMME LINJE FRA BIL TIL TANK FOR VANN
LD TR0
AND L21_VANN_T04_VANN
MOV(021) #30 L2_1_UT_VANN_PRS  ; PRS TOEMME LINJE FRA BIL TIL TANK FOR VANN
LD TR0
AND L21_VANN_T04_MELK
MOV(021) #30 L2_1_UT_VANN_PRS  ; PRS TOEMME LINJE FRA BIL TIL TANK FOR VANN
LD TR0
AND L21_VANN_T05_VANN
MOV(021) #30 L2_1_UT_VANN_PRS  ; PRS TOEMME LINJE FRA BIL TIL TANK FOR VANN
LD TR0
AND L21_VANN_T05_MELK
MOV(021) #30 L2_1_UT_VANN_PRS  ; PRS TOEMME LINJE FRA BIL TIL TANK FOR VANN
LD TR0
AND L21_MELK_T03_VANN
MOV(021) #30 L2_1_UT_VANN_PRS  ; PRS TOEMME LINJE FRA BIL TIL TANK FOR VANN
LD TR0
AND L21_MELK_T04_VANN
MOV(021) #300 L2_1_UT_VANN_PRS  ; PRS TOEMME LINJE FRA BIL TIL TANK FOR VANN
LD TR0
AND L21_MELK_T05_VANN
MOV(021) #30 L2_1_UT_VANN_PRS  ; PRS TOEMME LINJE FRA BIL TIL TANK FOR VANN
LD TR0
TIM 0684 L2_1_UT_VANN_PRS  ; PRS TOEMME LINJE FRA BIL TIL TANK FOR VANN, L2_1_VANN_DR_S

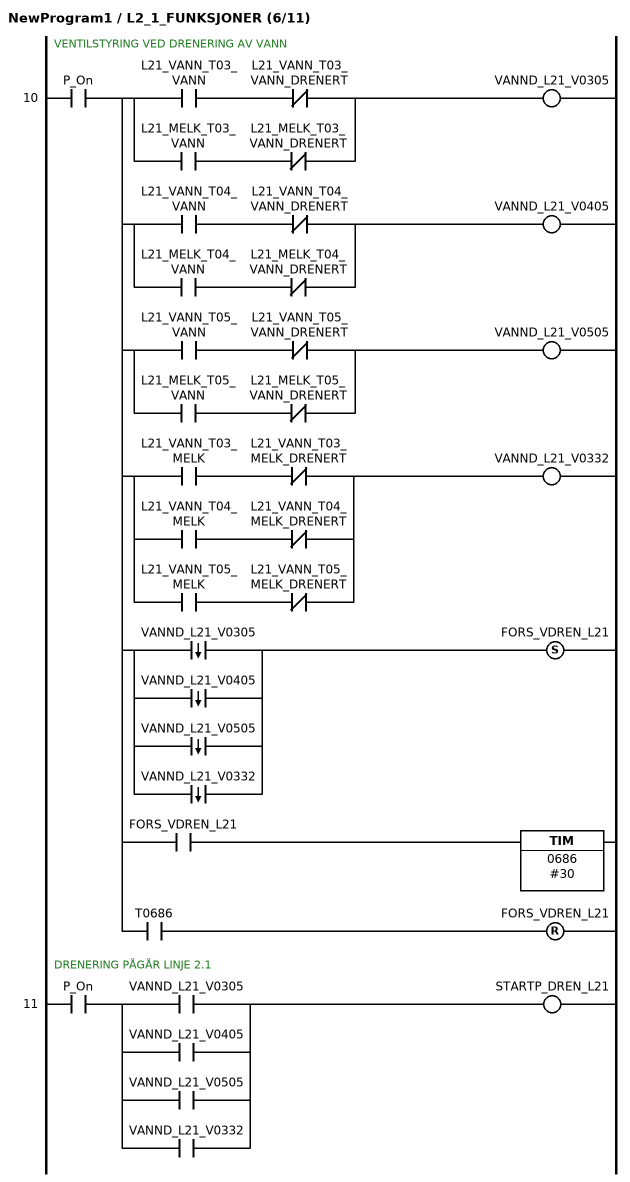
; rung 10: VENTILSTYRING VED DRENERING AV VANN
LD P_On
OUT TR0
LD L21_VANN_T03_VANN
ANDNOT L21_VANN_T03_VANN_DRENERT
LD L21_MELK_T03_VANN
ANDNOT L21_MELK_T03_VANN_DRENERT
ORLD
ANDLD
OUT VANND_L21_V0305
LD TR0
LD L21_VANN_T04_VANN
ANDNOT L21_VANN_T04_VANN_DRENERT
LD L21_MELK_T04_VANN
ANDNOT L21_MELK_T04_VANN_DRENERT
ORLD
ANDLD
OUT VANND_L21_V0405
LD TR0
LD L21_VANN_T05_VANN
ANDNOT L21_VANN_T05_VANN_DRENERT
LD L21_MELK_T05_VANN
ANDNOT L21_MELK_T05_VANN_DRENERT
ORLD
ANDLD
OUT VANND_L21_V0505
LD TR0
LD L21_VANN_T03_MELK
ANDNOT L21_VANN_T03_MELK_DRENERT
LD L21_VANN_T04_MELK
ANDNOT L21_VANN_T04_MELK_DRENERT
ORLD
LD L21_VANN_T05_MELK
ANDNOT L21_VANN_T05_MELK_DRENERT
ORLD
ANDLD
OUT VANND_L21_V0332
LD TR0
%LD VANND_L21_V0305
%OR VANND_L21_V0405
%OR VANND_L21_V0505
%OR VANND_L21_V0332
ANDLD
SET FORS_VDREN_L21
LD TR0
AND FORS_VDREN_L21
TIM 0686 #30
LD TR0
AND T0686
RSET FORS_VDREN_L21
; rung 11: DRENERING PÅGÅR LINJE 2.1
LD P_On
LD VANND_L21_V0305
OR VANND_L21_V0405
OR VANND_L21_V0505
OR VANND_L21_V0332
ANDLD
OUT STARTP_DREN_L21

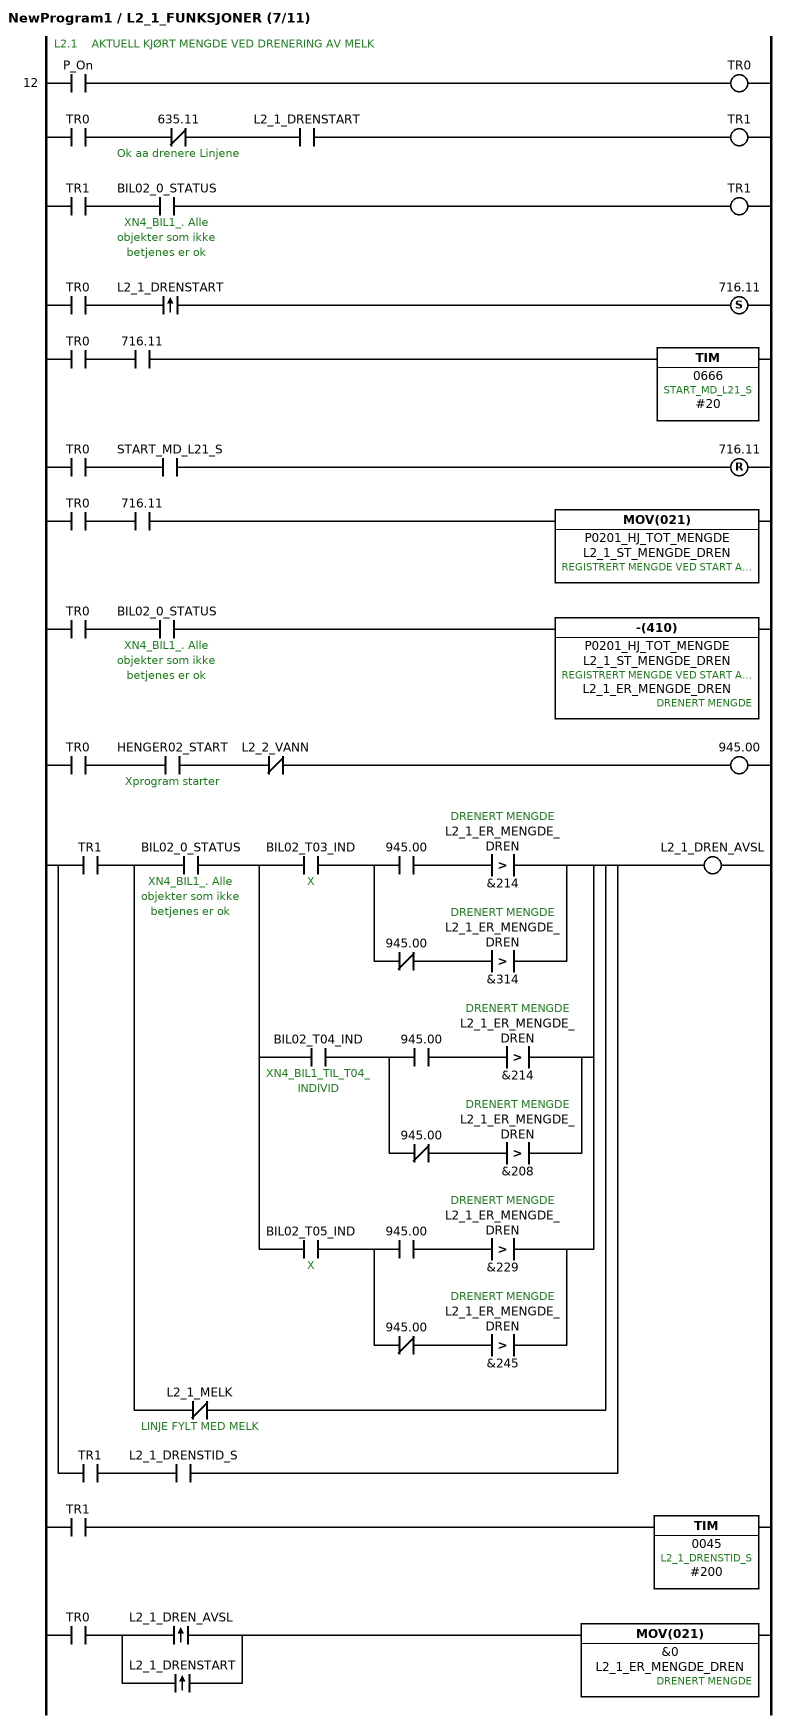
; rung 12: L2.1    AKTUELL KJØRT MENGDE VED DRENERING AV MELK
LD P_On
OUT TR0
@AND L2_1_DRENSTART
SET 716.11
LD TR0
AND 716.11
TIM 0666 #20  ; START_MD_L21_S
LD TR0
AND START_MD_L21_S
RSET 716.11
LD TR0
AND 716.11
MOV(021) P0201_HJ_TOT_MENGDE L2_1_ST_MENGDE_DREN  ; REGISTRERT MENGDE VED START AV DREN.
LD TR0
AND BIL02_0_STATUS  ; XN4_BIL1_. Alle objekter som ikke betjenes er ok
-(410) P0201_HJ_TOT_MENGDE L2_1_ST_MENGDE_DREN L2_1_ER_MENGDE_DREN  ; REGISTRERT MENGDE VED START AV DREN., DRENERT MENGDE
LD TR0
AND HENGER02_START  ; Xprogram starter
ANDNOT L2_2_VANN
OUT 945.00
LD TR0
ANDNOT 635.11  ; Ok aa drenere Linjene
AND L2_1_DRENSTART
OUT TR1
LD BIL02_0_STATUS  ; XN4_BIL1_. Alle objekter som ikke betjenes er ok
LD BIL02_T03_IND  ; X
LD 945.00
AND>(320) L2_1_ER_MENGDE_DREN &214  ; DRENERT MENGDE
LDNOT 945.00
AND>(320) L2_1_ER_MENGDE_DREN &314  ; DRENERT MENGDE
ORLD
ANDLD
LD BIL02_T04_IND  ; XN4_BIL1_TIL_T04_INDIVID
LD 945.00
AND>(320) L2_1_ER_MENGDE_DREN &214  ; DRENERT MENGDE
LDNOT 945.00
AND>(320) L2_1_ER_MENGDE_DREN &208  ; DRENERT MENGDE
ORLD
ANDLD
ORLD
LD BIL02_T05_IND  ; X
LD 945.00
AND>(320) L2_1_ER_MENGDE_DREN &229  ; DRENERT MENGDE
LDNOT 945.00
AND>(320) L2_1_ER_MENGDE_DREN &245  ; DRENERT MENGDE
ORLD
ANDLD
ORLD
ANDLD
ORNOT L2_1_MELK  ; LINJE FYLT MED MELK
ANDLD
LD TR1
AND BIL02_0_STATUS  ; XN4_BIL1_. Alle objekter som ikke betjenes er ok
OUT TR1
AND L2_1_DRENSTID_S
ORLD
OUT L2_1_DREN_AVSL
LD TR1
TIM 0045 #200  ; L2_1_DRENSTID_S
LD TR0
@LD L2_1_DREN_AVSL
@OR L2_1_DRENSTART
ANDLD
MOV(021) &0 L2_1_ER_MENGDE_DREN  ; DRENERT MENGDE

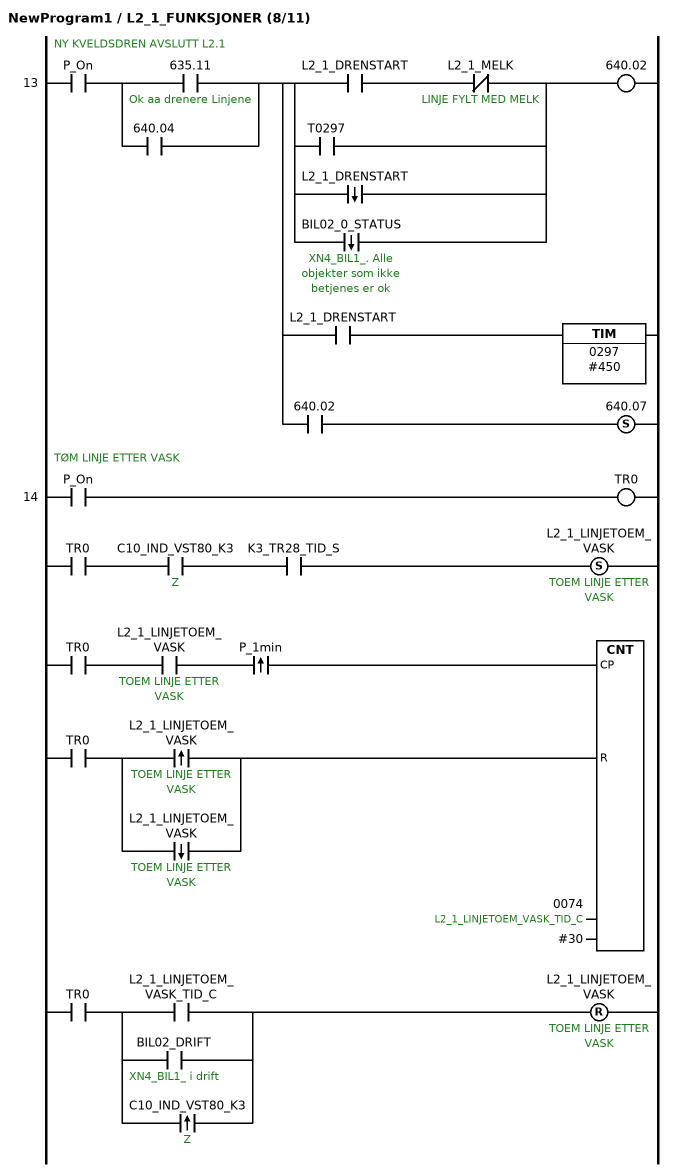
; rung 13: NY KVELDSDREN AVSLUTT L2.1
LD P_On
LD 635.11  ; Ok aa drenere Linjene
OR 640.04
ANDLD
OUT TR0
LD L2_1_DRENSTART
ANDNOT L2_1_MELK  ; LINJE FYLT MED MELK
OR T0297
%OR L2_1_DRENSTART
%OR BIL02_0_STATUS  ; XN4_BIL1_. Alle objekter som ikke betjenes er ok
ANDLD
OUT 640.02
LD TR0
AND L2_1_DRENSTART
TIM 0297 #450
LD TR0
AND 640.02
SET 640.07
; rung 14: TØM LINJE ETTER VASK
LD P_On
OUT TR0
AND C10_IND_VST80_K3  ; Z
AND K3_TR28_TID_S
SET L2_1_LINJETOEM_VASK  ; TOEM LINJE ETTER VASK
LD TR0
AND L2_1_LINJETOEM_VASK  ; TOEM LINJE ETTER VASK
@AND P_1min
LD TR0
@LD L2_1_LINJETOEM_VASK  ; TOEM LINJE ETTER VASK
%OR L2_1_LINJETOEM_VASK  ; TOEM LINJE ETTER VASK
ANDLD
CNT 0074 #30  ; L2_1_LINJETOEM_VASK_TID_C
LD TR0
LD L2_1_LINJETOEM_VASK_TID_C
OR BIL02_DRIFT  ; XN4_BIL1_ i drift
@OR C10_IND_VST80_K3  ; Z
ANDLD
RSET L2_1_LINJETOEM_VASK  ; TOEM LINJE ETTER VASK

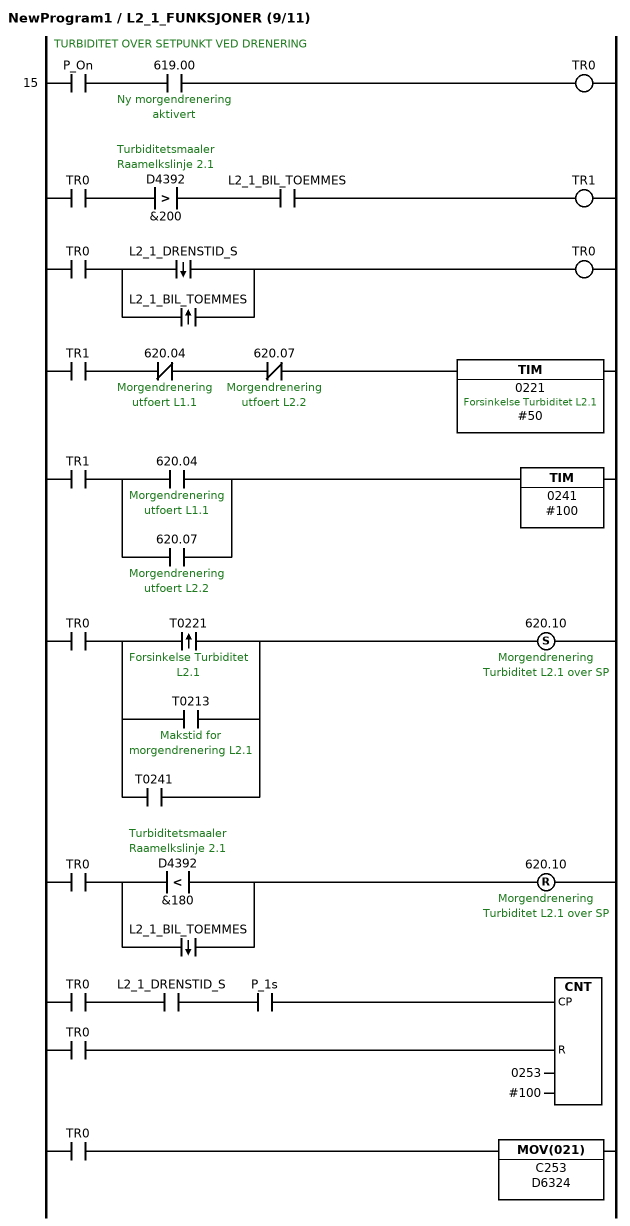
; rung 15: TURBIDITET OVER SETPUNKT VED DRENERING
LD P_On
AND 619.00  ; Ny morgendrenering aktivert
OUT TR0
AND>(320) D4392 &200  ; Turbiditetsmaaler Raamelkslinje 2.1
AND L2_1_BIL_TOEMMES
OUT TR1
ANDNOT 620.04  ; Morgendrenering utfoert L1.1
ANDNOT 620.07  ; Morgendrenering utfoert L2.2
TIM 0221 #50  ; Forsinkelse Turbiditet L2.1
LD TR1
LD 620.04  ; Morgendrenering utfoert L1.1
OR 620.07  ; Morgendrenering utfoert L2.2
ANDLD
TIM 0241 #100
LD TR0
@LD T0221  ; Forsinkelse Turbiditet L2.1
OR T0213  ; Makstid for morgendrenering L2.1
OR T0241
ANDLD
SET 620.10  ; Morgendrenering Turbiditet L2.1 over SP
LD TR0
LD<(310) D4392 &180  ; Turbiditetsmaaler Raamelkslinje 2.1
%OR L2_1_BIL_TOEMMES
ANDLD
RSET 620.10  ; Morgendrenering Turbiditet L2.1 over SP
LD TR0
AND L2_1_DRENSTID_S
AND P_1s
LD TR0
%LD L2_1_DRENSTID_S
@OR L2_1_BIL_TOEMMES
ANDLD
OUT TR0
CNT 0253 #100
LD TR0
MOV(021) C253 D6324

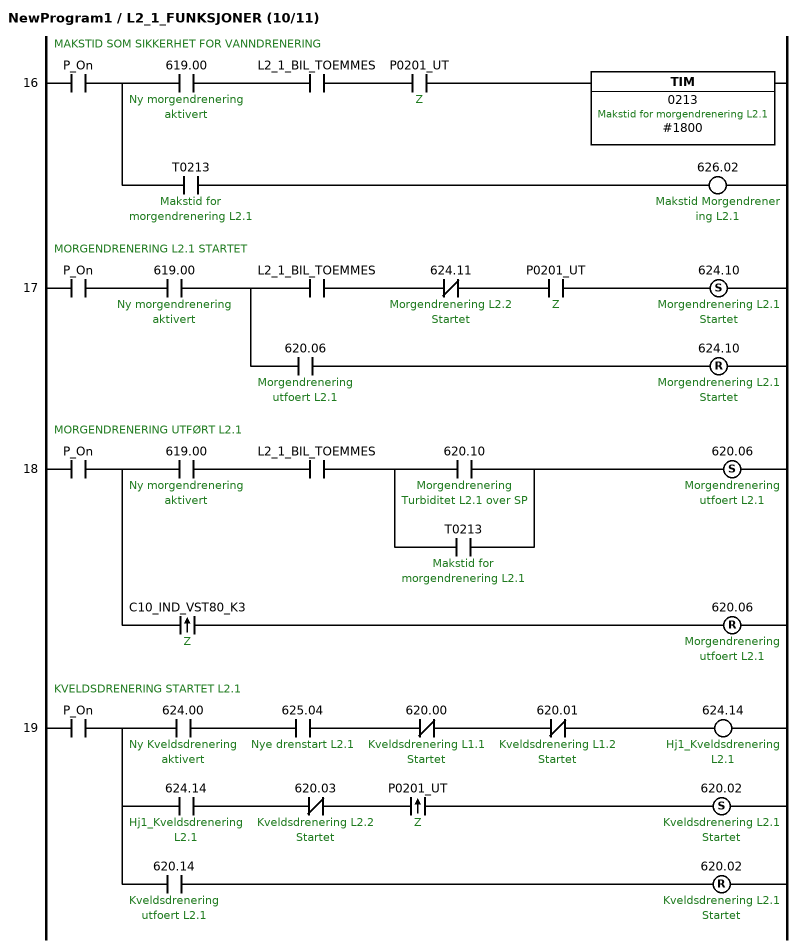
; rung 16: MAKSTID SOM SIKKERHET FOR VANNDRENERING
LD P_On
OUT TR0
AND 619.00  ; Ny morgendrenering aktivert
AND L2_1_BIL_TOEMMES
AND P0201_UT  ; Z
TIM 0213 #1800  ; Makstid for morgendrenering L2.1
LD TR0
AND T0213  ; Makstid for morgendrenering L2.1
OUT 626.02  ; Makstid Morgendrenering L2.1
; rung 17: MORGENDRENERING L2.1 STARTET
LD P_On
AND 619.00  ; Ny morgendrenering aktivert
OUT TR0
AND L2_1_BIL_TOEMMES
ANDNOT 624.11  ; Morgendrenering L2.2 Startet
AND P0201_UT  ; Z
SET 624.10  ; Morgendrenering L2.1 Startet
LD TR0
AND 620.06  ; Morgendrenering utfoert L2.1
RSET 624.10  ; Morgendrenering L2.1 Startet
; rung 18: MORGENDRENERING UTFØRT L2.1
LD P_On
OUT TR0
AND 619.00  ; Ny morgendrenering aktivert
AND L2_1_BIL_TOEMMES
LD 620.10  ; Morgendrenering Turbiditet L2.1 over SP
OR T0213  ; Makstid for morgendrenering L2.1
ANDLD
SET 620.06  ; Morgendrenering utfoert L2.1
LD TR0
@AND C10_IND_VST80_K3  ; Z
RSET 620.06  ; Morgendrenering utfoert L2.1
; rung 19: KVELDSDRENERING STARTET L2.1
LD P_On
OUT TR0
AND 624.00  ; Ny Kveldsdrenering aktivert
AND 625.04  ; Nye drenstart L2.1
ANDNOT 620.00  ; Kveldsdrenering L1.1 Startet
ANDNOT 620.01  ; Kveldsdrenering L1.2 Startet
OUT 624.14  ; Hj1_Kveldsdrenering L2.1
LD TR0
AND 624.14  ; Hj1_Kveldsdrenering L2.1
ANDNOT 620.03  ; Kveldsdrenering L2.2 Startet
@AND P0201_UT  ; Z
SET 620.02  ; Kveldsdrenering L2.1 Startet
LD TR0
AND 620.14  ; Kveldsdrenering utfoert L2.1
RSET 620.02  ; Kveldsdrenering L2.1 Startet

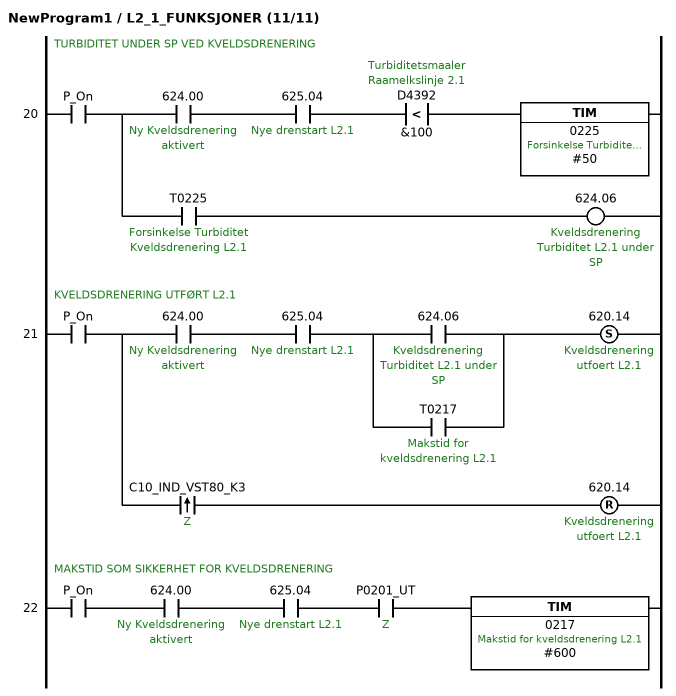
; rung 20: TURBIDITET UNDER SP VED KVELDSDRENERING
LD P_On
OUT TR0
AND 624.00  ; Ny Kveldsdrenering aktivert
AND 625.04  ; Nye drenstart L2.1
AND<(310) D4392 &100  ; Turbiditetsmaaler Raamelkslinje 2.1
TIM 0225 #50  ; Forsinkelse Turbiditet Kveldsdrenering L2.1
LD TR0
AND T0225  ; Forsinkelse Turbiditet Kveldsdrenering L2.1
OUT 624.06  ; Kveldsdrenering Turbiditet L2.1 under SP
; rung 21: KVELDSDRENERING UTFØRT L2.1
LD P_On
OUT TR0
AND 624.00  ; Ny Kveldsdrenering aktivert
AND 625.04  ; Nye drenstart L2.1
LD 624.06  ; Kveldsdrenering Turbiditet L2.1 under SP
OR T0217  ; Makstid for kveldsdrenering L2.1
ANDLD
SET 620.14  ; Kveldsdrenering utfoert L2.1
LD TR0
@AND C10_IND_VST80_K3  ; Z
RSET 620.14  ; Kveldsdrenering utfoert L2.1
; rung 22: MAKSTID SOM SIKKERHET FOR KVELDSDRENERING
LD P_On
AND 624.00  ; Ny Kveldsdrenering aktivert
AND 625.04  ; Nye drenstart L2.1
AND P0201_UT  ; Z
TIM 0217 #600  ; Makstid for kveldsdrenering L2.1
; rung 23: Ingen_kommentar_funnet

### Section L2_2_STATUS

